(* CODESYS project SPT_NCI.library
   Version: 4.0.0
   Title: SPT NCI
   DefaultNamespace: SPT_NCI
   Placeholder: SPT NCI
   Company: Beckhoff Automation LLC

Project tree, tasks and I/O mapping:
  libraries: SPT Base Types, * (Beckhoff Automation LLC); SPT Event Logger, * (Beckhoff Automation LLC); Tc2_NCI, * (Beckhoff Automation GmbH); Tc2_Standard, * (Beckhoff Automation GmbH); Tc2_System, * (Beckhoff Automation GmbH); Tc3_EventLogger, * (Beckhoff Automation GmbH); Tc3_Module, * (Beckhoff Automation GmbH)
  DUTs/
    data type ST_NciBase_Command
    data type ST_NciBase_Config
    data type ST_NciBase_HMI
    data type ST_NciBase_Status
    data type ST_NciChannel
  FunctionBlocks/
    function block FB_Component_NciBase [ST]: Reset, CyclicLogic, BlockSearch, BuildNciGroup, ConfirmHsk, DissolveNciGroup, EnableRetrace, InterpreterStart, InterpreterStop, InterpreterStopOnPath, IsFastMFunction, LoadNciProgram, ResumeAfterEstop, RetraceBackward, RetraceForward, SetSearchOptionFlags, StepOnAfterBlocksearch, BlockSearchStartPosition, Channel, Deceleration, GetHskMFunction, GroupIsBuilt, InterpreterState, IsHandshake, Jerk, Override, ProgramPath, CreateEvents, HMICommunication, Monitoring, Q1AxisId, Q2AxisId, Q3AxisId, Q4AxisId, Q5AxisId, XAxisId, YAxisId, ZAxisId, Initialize
    function block FB_Component_NciParameterBase [ST]: Reset, CyclicLogic, CreateEvents, Channel, Initialize
    function block FB_Component_NciReadWriteRParameter [ST]: Reset, CyclicLogic, Monitoring, Read, Write
  Interfaces/
    interface I_NciBase: BlockSearch, BuildNciGroup, ConfirmHsk, DissolveNciGroup, EnableRetrace, InterpreterStart, InterpreterStop, InterpreterStopOnPath, IsFastMFunction, LoadNciProgram, ResumeAfterEstop, RetraceBackward, RetraceForward, SetSearchOptionFlags, StepOnAfterBlocksearch, BlockSearchStartPosition, Deceleration, GetHskMFunction, GroupIsBuilt, InterpreterState, IsHandshake, Jerk, Override, ProgramPath
    interface I_NciChannel: Channel
  Project Information/
    function F_GetCompany [ST]
    function F_GetTitle [ST]
    function F_GetVersion [ST]
  Utilities/
    function F_ADSErrorCodeExt [ST]
  Version/
    global variables Global_Version
  00000000-0000-0000-0000-000000000000|LICENSE
  LICENSE
*)

// DUTs/ST_NciBase_Command
TYPE ST_NciBase_Command :
	STRUCT
		BuildGroup		   : BOOL;
		DissolveGroup	   : BOOL;
		LoadNciProgram	   : BOOL;
		ItpStart		   : BOOL;
		ItpStop			   : BOOL;
		ItpEstopStopOnPath : BOOL;
		Resume			   : BOOL;
		SetOverride		   : BOOL;
		Override		   : UDINT; //Override in 0..1000000 (0..100%)
	END_STRUCT
END_TYPE

// DUTs/ST_NciBase_Config
TYPE ST_NciBase_Config :
	STRUCT
	END_STRUCT
END_TYPE

// DUTs/ST_NciBase_HMI
TYPE ST_NciBase_HMI :
	STRUCT
		Config	: ST_NciBase_Config;
		Command : ST_NciBase_Command;
		Status	: ST_NciBase_Status;
	END_STRUCT
END_TYPE

// DUTs/ST_NciBase_Status
TYPE ST_NciBase_Status :
	STRUCT
		NcToPlc : NCTOPLC_NCICHANNEL_REF;
	END_STRUCT
END_TYPE

// DUTs/ST_NciChannel
TYPE ST_NciChannel :
	STRUCT
		NcToPLC AT %I* : NCTOPLC_NCICHANNEL_REF;
		PlcToNc AT %Q* : PLCTONC_NCICHANNEL_REF;
	END_STRUCT
END_TYPE

// Version/Global_Version
{attribute 'TcGenerated'}
{attribute 'no-analysis'}
{attribute 'linkalways'}

// This function has been automatically generated from the project information.
VAR_GLOBAL CONSTANT
	{attribute 'const_non_replaced'}
	stLibVersion_SPT_NCI : ST_LibVersion := (iMajor := 4, iMinor := 0, iBuild := 0, iRevision := 0, nFlags := 0, sVersion := '4.0.0');
END_VAR

// FunctionBlocks/FB_Component_NciBase
FUNCTION_BLOCK FB_Component_NciBase EXTENDS FB_ComponentBase IMPLEMENTS I_NciBase
VAR
	// Channel connection
	NciChannel : ST_NciChannel;

	// Properties
	_ProgramPath		   : STRING := 'C:\TwinCAT\Mc\Nci\9999.nc';
	_XAxisId			   : UDINT	:= 0;
	_YAxisId			   : UDINT	:= 0;
	_ZAxisId			   : UDINT	:= 0;
	_Q1AxisId			   : UDINT	:= 0;
	_Q2AxisId			   : UDINT	:= 0;
	_Q3AxisId			   : UDINT	:= 0;
	_Q4AxisId			   : UDINT	:= 0;
	_Q5AxisId			   : UDINT	:= 0;
	_GroupIsBuilt		   : BOOL;
	_Jerk				   : LREAL;
	_Deceleration		   : LREAL;
	_BlockSearchOptionFlag : ST_ItpBlockSearchOptions := (bScanStartPos := TRUE);
	_StartPosition		   : ST_ItpBlockSearchStartPosition;

	// Internal Variables
	BuildGroup		 : CfgBuildExt3DGroup;
	DissolveGroup	 : CfgReconfigGroup;
	ResetNci		 : ItpResetEx2;
	LoadProgram		 : ItpLoadProgEx;
	StartStop		 : ItpStartStopEx;
	EStopOnPath		 : ItpEstopEx;
	StepOnAfterEStop : ItpStepOnAfterEStopEx;
	ResetFastMCode	 : ItpResetFastMFuncEx;
	ConfirmHandshake : ItpConfirmHsk;

	// Retrace functions
	EnableFeederBackup	: ItpEnableFeederBackup;
	RetraceMoveBackward : ItpRetraceMoveBackward;
	RetraceMoveForward	: ItpRetraceMoveForward;

	// Blocksearch
	InterpreterBlockSearch : ItpBlocksearch;
	BlockOn				   : ItpStepOnAfterBlocksearch;

	// HMI
	NciBase_HMI : ST_NciBase_HMI;

	// Alarms
	ComponentNciBaseAlarms : ARRAY[1..COMPONENT_NCI_BASE_ALARM_COUNT] OF FB_TcAlarm;
END_VAR

VAR CONSTANT
	COMPONENT_NCI_BASE_ALARM_COUNT : UDINT := 12;
END_VAR

// Clears error flags and error IDs for this component
METHOD PUBLIC Reset : BOOL
F_ClearAllEventsInClass(ComponentNciBaseAlarms);
_Error			  := FALSE;
_ErrorId		  := 0;
ResetNci.bExecute := TRUE;
Reset			  := SUPER^.Reset();
END_METHOD

// This method serves as the entry point for all underlying FB logic
METHOD PUBLIC CyclicLogic

// This method should be called cyclically by descendant function blocks by invoking SUPER^.CyclicLogic().  Alternatively, the contents of this method could be reimplemented entirely in which case a call to this method would not be necessary.
IF NOT _InitComplete THEN
	_InitComplete := Initialize();
	RETURN;
END_IF

(* NCI FBs *)

// Build NCI Group
BuildGroup(nGroupId := NciChannel.NcToPLC.GrpId, tTimeout := T#1S);
IF BuildGroup.bErr AND BuildGroup.bExecute THEN
	_GroupIsBuilt := FALSE;
	_Error		  := TRUE;
	_ErrorId	  := BuildGroup.nErrId;
END_IF

IF NOT BuildGroup.bBusy THEN
	BuildGroup.bExecute := FALSE;
END_IF

// Dissolve NCI Group
DissolveGroup(nGroupId := NciChannel.NcToPLC.GrpId, tTimeOut := T#1S);
IF DissolveGroup.bErr AND DissolveGroup.bExecute THEN
	_Error	 := TRUE;
	_ErrorId := DissolveGroup.nErrId;
END_IF

IF NOT DissolveGroup.bBusy THEN
	DissolveGroup.bExecute := FALSE;
END_IF

// Reset
ResetNci(sNciToPlc := NciChannel.NcToPlc, tTimeOut := T#1S);
IF ResetNci.bErr AND ResetNci.bExecute THEN
	_Error	 := TRUE;
	_ErrorId := ResetNci.nErrId;
END_IF

IF NOT ResetNci.bBusy THEN
	ResetNci.bExecute := FALSE;
END_IF

// Load Program
LoadProgram(sNciToPlc := NciChannel.NcToPLC,
			sPrg	  := _ProgramPath,
			nLength	  := INT_TO_UDINT(LEN(_ProgramPath)),
			tTimeOut  := T#1S);

IF LoadProgram.bErr AND LoadProgram.bExecute THEN
	_Error	 := TRUE;
	_ErrorId := LoadProgram.nErrId;
END_IF

IF NOT LoadProgram.bBusy THEN
	LoadProgram.bExecute := FALSE;
END_IF

// Start/Stop Interpreter
StartStop(sNciToPlc := NciChannel.NcToPLC, tTimeOut := T#1S);
IF StartStop.bErr AND (StartStop.bStop OR StartStop.bStart) THEN
	_Error	 := TRUE;
	_ErrorId := StartStop.nErrId;
END_IF

IF NOT StartStop.bBusy THEN
	StartStop.bStop	 := FALSE;
	StartStop.bStart := FALSE;
END_IF

//
EStopOnPath(sNciToPlc := NciChannel.NcToPLC,
			fDec	  := _Deceleration,
			fJerk	  := _Jerk,
			tTimeOut  := T#1S);

IF EStopOnPath.bErr AND EStopOnPath.bExecute THEN
	_Error	 := TRUE;
	_ErrorId := EStopOnPath.nErrId;
END_IF

IF NOT EStopOnPath.bBusy THEN
	EStopOnPath.bExecute := FALSE;
END_IF

StepOnAfterEStop(sNciToPlc := NciChannel.NcToPLC, tTimeOut := T#1S);
IF StepOnAfterEStop.bErr AND StepOnAfterEStop.bExecute THEN
	_Error	 := TRUE;
	_ErrorId := StepOnAfterEStop.nErrId;
END_IF

IF NOT StepOnAfterEStop.bBusy THEN
	StepOnAfterEStop.bExecute := FALSE;
END_IF

// Retracing
EnableFeederBackup(bEnable := TRUE, tTimeOut := T#1S, sNciToPlc := NciChannel.NcToPLC);
IF EnableFeederBackup.bErr AND EnableFeederBackup.bExecute THEN
	_Error	 := TRUE;
	_ErrorId := EnableFeederBackup.nErrId;
END_IF

IF NOT EnableFeederBackup.bBusy THEN
	EnableFeederBackup.bExecute := FALSE;
END_IF

RetraceMoveBackward(sNciToPlc := NciChannel.NcToPLC);
IF RetraceMoveBackward.bErr AND RetraceMoveBackward.bExecute THEN
	_Error	 := TRUE;
	_ErrorId := RetraceMoveBackward.nErrId;
END_IF

IF NOT RetraceMoveBackward.bBusy THEN
	RetraceMoveBackward.bExecute := FALSE;
END_IF

RetraceMoveForward(sNciToPlc := NciChannel.NcToPLC);
IF RetraceMoveForward.bErr AND RetraceMoveForward.bExecute THEN
	_Error	 := TRUE;
	_ErrorId := RetraceMoveForward.nErrId;
END_IF

IF NOT RetraceMoveForward.bBusy THEN
	RetraceMoveForward.bExecute := FALSE;
END_IF

// Blocksearch
InterpreterBlockSearch(sPrgName		  := _ProgramPath,
					   nPrgLength	  := INT_TO_UDINT(LEN(_ProgramPath)),
					   tTimeOut		  := T#5S,
					   sAxesList	  :=,
					   sOptions		  := _BlockSearchOptionFlag,
					   sStartPosition => _StartPosition,
					   sNciToPlc	  := NciChannel.NcToPLC);

IF InterpreterBlockSearch.bErr AND InterpreterBlockSearch.bExecute THEN
	_Error	 := TRUE;
	_ErrorId := InterpreterBlockSearch.nErrId;
END_IF

IF NOT InterpreterBlockSearch.bBusy THEN
	InterpreterBlockSearch.bExecute := FALSE;
END_IF

BlockOn(sNciToPlc := NciChannel.NcToPLC, tTimeOut := T#1S);
IF BlockOn.bErr AND BlockOn.bExecute THEN
	_Error	 := TRUE;
	_ErrorId := BlockOn.nErrId;
END_IF

IF NOT BlockOn.bBusy THEN
	BlockOn.bExecute := FALSE;
END_IF

// MCode
ResetFastMCode(sNciToPlc := NciChannel.NcToPLC, tTimeOut := T#1S);
ResetFastMCode.bExecute := FALSE;
ConfirmHandshake(sNciToPlc := NciChannel.NcToPlc, sPlcToNci := NciChannel.PlcToNc);
ConfirmHandshake.bExecute := FALSE;

// Busy
_Busy := ResetNci.bBusy OR DissolveGroup.bBusy OR BuildGroup.bBusy OR EnableFeederBackup.bBusy OR EStopOnPath.bBusy OR RetraceMoveForward.bBusy OR RetraceMoveBackward.bBusy OR InterpreterBlockSearch.bBusy OR BlockOn.bBusy;

// Call Super
SUPER^.CyclicLogic();
_CurrentAlarmSeverity := F_GetMaxSeverityRaised(Alarms := ComponentNciBaseAlarms, CurrentSeverity := _CurrentAlarmSeverity);
END_METHOD

METHOD BlockSearch : BOOL
VAR_INPUT
	BlockId			: UINT;
	BlockSearchMode : E_ItpBlockSearchMode;
	DryRunMode		: E_ItpDryRunMode;
	LineLength		: UDINT;
END_VAR
IF _Busy OR _Error THEN
	RETURN;
END_IF

InterpreterBlockSearch.nBlockId			:= BlockId;
InterpreterBlockSearch.eBlockSearchMode := BlockSearchMode;
InterpreterBlockSearch.eDryRunMode		:= DryRunMode;
InterpreterBlockSearch.fLength			:= LineLength;
InterpreterBlockSearch.bExecute			:= TRUE;
BlockSearch								:= TRUE;
END_METHOD

METHOD PUBLIC BuildNciGroup : BOOL
IF _Busy OR _Error THEN
	RETURN;
END_IF

BuildGroup.nXAxisId	 := _XAxisId;
BuildGroup.nYAxisId	 := _YAxisId;
BuildGroup.nZAxisId	 := _ZAxisId;
BuildGroup.nQ1AxisId := _Q1AxisId;
BuildGroup.nQ2AxisId := _Q2AxisId;
BuildGroup.nQ3AxisId := _Q3AxisId;
BuildGroup.nQ4AxisId := _Q4AxisId;
BuildGroup.nQ5AxisId := _Q5AxisId;
BuildGroup.bExecute	 := TRUE;
_GroupIsBuilt		 := TRUE;
BuildNciGroup		 := TRUE;
END_METHOD

METHOD ConfirmHsk : BOOL
VAR_INPUT
END_VAR
ConfirmHandshake.bExecute := TRUE;
ConfirmHsk				  := TRUE;
END_METHOD

METHOD PUBLIC DissolveNciGroup : BOOL
IF _Busy THEN
	RETURN;
END_IF

_GroupIsBuilt		   := FALSE;
DissolveGroup.bExecute := TRUE;
DissolveNciGroup	   := TRUE;
END_METHOD

METHOD EnableRetrace : BOOL
VAR_INPUT
END_VAR
IF _Busy OR _Error THEN
	RETURN;
END_IF

EnableFeederBackup.bExecute := TRUE;
EnableRetrace				:= TRUE;
END_METHOD

METHOD InterpreterStart : BOOL
IF _Busy OR _Error THEN
	RETURN;
END_IF

StartStop.bStart := TRUE;
InterpreterStart := TRUE;
END_METHOD

METHOD InterpreterStop : BOOL
StartStop.bStop := TRUE;
InterpreterStop := TRUE;
END_METHOD

METHOD InterpreterStopOnPath : BOOL
VAR_INPUT
END_VAR
EStopOnPath.bExecute  := TRUE;
InterpreterStopOnPath := TRUE;
END_METHOD

METHOD IsFastMFunction : BOOL
VAR_INPUT
	M		  : INT;
	AutoReset : BOOL; // Reset MCode at next cycle
END_VAR
IsFastMFunction := ItpIsFastMFunc(NFastMfuncNo := M, NciChannel.NcToPlc);
IF IsFastMfunction AND AutoReset THEN
	ResetFastMCode.nMFuncNo := TO_UINT(M);
	ResetFastMCode.bExecute := TRUE;
END_IF
END_METHOD

METHOD LoadNciProgram : BOOL
IF _Busy THEN
	RETURN;
END_IF

IF _ProgramPath = '' THEN
	TRACE('NCI Program can not be loaded, Path is empty!');
END_IF

LoadProgram.bExecute := TRUE;
LoadNciProgram		 := TRUE;
END_METHOD

// Resume after stop on patch (ItpEstopEx)
METHOD ResumeAfterEstop : BOOL
VAR_INPUT
END_VAR
IF _Busy OR _Error THEN
	RETURN;
END_IF

StepOnAfterEStop.bExecute := TRUE;
ResumeAfterEstop		  := TRUE;
END_METHOD

METHOD RetraceBackward : BOOL
VAR_INPUT
END_VAR
IF _Busy OR _Error THEN
	RETURN;
END_IF

RetraceMoveBackward.bExecute := TRUE;
RetraceBackward				 := TRUE;
END_METHOD

METHOD RetraceForward : BOOL
VAR_INPUT
END_VAR
IF _Busy OR _Error THEN
	RETURN;
END_IF

RetraceMoveForward.bExecute := TRUE;
RetraceForward				:= TRUE;
END_METHOD

METHOD SetSearchOptionFlags
VAR_INPUT
	IsRetrace		  : BOOL;
	IsRetraceBackward : BOOL;
	ScanStartPos	  : BOOL;
END_VAR
_BlockSearchOptionFlag.bIsRetrace		:= IsRetrace;
_BlockSearchOptionFlag.bRetraceBackward := IsRetraceBackward;
_BlockSearchOptionFlag.bScanStartPos	:= ScanStartPos;
END_METHOD

METHOD StepOnAfterBlocksearch : BOOL
VAR_INPUT
END_VAR
IF _Busy OR _Error THEN
	RETURN;
END_IF

BlockOn.bExecute	   := TRUE;
StepOnAfterBlocksearch := TRUE;
END_METHOD

PROPERTY BlockSearchStartPosition : ST_ItpBlockSearchStartPosition
GET
BlockSearchStartPosition := _StartPosition;
END_GET
END_PROPERTY

PROPERTY Channel : REFERENCE TO ST_NciChannel
GET
Channel REF= NciChannel;
END_GET
END_PROPERTY

PROPERTY Deceleration : LREAL
SET
_Deceleration := Deceleration;
END_SET
END_PROPERTY

PROPERTY GetHskMFunction : INT
GET
GetHskMFunction := ItpGetHskMFunc(NciChannel.NcToPLC);
END_GET
END_PROPERTY

PROPERTY GroupIsBuilt : BOOL
GET
GroupIsBuilt := _GroupIsBuilt;
END_GET
END_PROPERTY

// Use to query e.g. Tc2_NCI.NCI_INTERPRETER_READY
PROPERTY InterpreterState : UINT
GET
InterpreterState := NciChannel.NcToPLC.ItpState;
END_GET
END_PROPERTY

PROPERTY IsHandshake : BOOL
GET
IsHandshake := ItpIsHskMFunc(NciChannel.NcToPLC);
END_GET
END_PROPERTY

PROPERTY Jerk : LREAL
SET
_Jerk := Jerk;
END_SET
END_PROPERTY

// Override in 0..1000000 //Assigns override to all channel overrides, individual access via property channel.
PROPERTY Override : UDINT
SET
IF Override < 0 THEN
	NciChannel.PlcToNc.ChnAxesOvr	 := 0;
	NciChannel.PlcToNc.ChnSpindleOvr := 0;
ELSIF Override > 1_000_000 THEN
	NciChannel.PlcToNc.ChnAxesOvr	 := 1_000_000;
	NciChannel.PlcToNc.ChnSpindleOvr := 1_000_000;
ELSE
	NciChannel.PlcToNc.ChnAxesOvr	 := Override;
	NciChannel.PlcToNc.ChnSpindleOvr := Override;
END_IF
END_SET
END_PROPERTY

PROPERTY ProgramPath : STRING
GET
ProgramPath := _ProgramPath;
END_GET
SET
_ProgramPath := ProgramPath;
END_SET
END_PROPERTY

// Initializes event function blocks using this components's name
METHOD PROTECTED CreateEvents

// This method is called by Initialize() as required
SUPER^.CreateEvents();
F_CreateAllEventsInClass(Alarms		:= ComponentNciBaseAlarms,
						 ClassSize	:= SIZEOF(TC_EVENTS.NciAlarms),
						 pInitEvent := ADR(TC_EVENTS.NciAlarms.InitReferenceEvent),
						 Prefix		:= _Name);
END_METHOD

// Provides interlocks for HMI control and updates HMI status information for this component
METHOD PROTECTED HMICommunication
// This method is called cyclically by CyclicLogic()
VAR_INST
	HMICommandNciBase_RT : R_TRIG;
END_VAR
SUPER^.HMICommunication();
HMICommandNciBase_RT(CLK := (ComponentBase_HMI.Status.HMIControlAvailable AND NOT HMICommandActive_Base) AND (NciBase_HMI.Command.BuildGroup XOR NciBase_HMI.Command.DissolveGroup XOR NciBase_HMI.Command.LoadNciProgram XOR NciBase_HMI.Command.ItpStart XOR NciBase_HMI.Command.ItpStop XOR NciBase_Hmi.Command.ItpEstopStopOnPath XOR NciBase_Hmi.Command.Resume));

//Desendant components should observe this to interlock HMI commands
HMICommandActive_Descendant := ComponentBase_HMI.Status.HMIControlAvailable AND (NciBase_HMI.Command.BuildGroup OR NciBase_HMI.Command.DissolveGroup OR NciBase_HMI.Command.LoadNciProgram OR NciBase_HMI.Command.ItpStart OR NciBase_HMI.Command.ItpStop OR NciBase_Hmi.Command.ItpEstopStopOnPath OR NciBase_Hmi.Command.Resume);
IF HMICommandNciBase_RT.Q THEN
	IF NciBase_HMI.Command.BuildGroup THEN
		BuildNciGroup();
	END_IF

	IF NciBase_HMI.Command.DissolveGroup THEN
		DissolveNciGroup();
	END_IF

	IF NciBase_HMI.Command.LoadNciProgram THEN
		LoadNciProgram();
	END_IF

	IF NciBase_HMI.Command.ItpStart THEN
		InterpreterStart();
	END_IF

	IF NciBase_HMI.Command.ItpStop THEN
		InterpreterStop();
	END_IF

	IF NciBase_Hmi.Command.ItpEstopStopOnPath THEN
		InterpreterStopOnPath();
	END_IF

	IF NciBase_Hmi.Command.Resume THEN
		ResumeAfterEstop();
	END_IF
END_IF

NciBase_HMI.Command.BuildGroup		   := FALSE;
NciBase_HMI.Command.DissolveGroup	   := FALSE;
NciBase_HMI.Command.LoadNciProgram	   := FALSE;
NciBase_HMI.Command.ItpStart		   := FALSE;
NciBase_HMI.Command.ItpStop			   := FALSE;
NciBase_Hmi.Command.ItpEstopStopOnPath := FALSE;
NciBase_Hmi.Command.Resume			   := FALSE;

// Set Override
IF NciBase_Hmi.Command.SetOverride THEN
	Override						:= NciBase_Hmi.Command.Override;
	NciBase_Hmi.Command.SetOverride := FALSE;
END_IF

// Status
NciBase_Hmi.Status.NcToPlc := NciChannel.NcToPlc;
END_METHOD

// Provides basic error detection and event handling for this component
METHOD PROTECTED Monitoring
VAR_INST
	RTrigError	: R_TRIG; // Error active - Error Bit remains On in NCI Fbs until new command is issued
	TempMessage : STRING;
END_VAR

// This method is called cyclically by CyclicLogic()
SUPER^.Monitoring();
RTrigError(CLK := _Error);
IF RTrigError.Q THEN
	// Build Group
	IF BuildGroup.bErr AND NOT ComponentNciBaseAlarms[E_NciAlarms.BuildGroup].bRaised THEN
		RaiseAlarmWithStrings(ComponentNciBaseAlarms[E_NciAlarms.BuildGroup], F_ADSErrorCodeExt(_ErrorId), '');
	END_IF

	// Load Program
	IF LoadProgram.bErr AND NOT ComponentNciBaseAlarms[E_NciAlarms.LoadProgram].bRaised THEN
		RaiseAlarmWithStrings(ComponentNciBaseAlarms[E_NciAlarms.LoadProgram], F_ADSErrorCodeExt(_ErrorId), '');
	END_IF

	// Start/ Stop
	IF EStopOnPath.bErr AND NOT ComponentNciBaseAlarms[E_NciAlarms.StopOnPath].bRaised THEN
		RaiseAlarmWithStrings(ComponentNciBaseAlarms[E_NciAlarms.StopOnPath], F_ADSErrorCodeExt(_ErrorId), '');
	END_IF

	IF StartStop.bErr AND NOT ComponentNciBaseAlarms[E_NciAlarms.StartStop].bRaised THEN
		RaiseAlarmWithStrings(ComponentNciBaseAlarms[E_NciAlarms.StartStop], F_ADSErrorCodeExt(_ErrorId), '');
	END_IF

	IF StepOnAfterEStop.bErr AND NOT ComponentNciBaseAlarms[E_NciAlarms.StepOnAfterEStop].bRaised THEN
		RaiseAlarmWithStrings(ComponentNciBaseAlarms[E_NciAlarms.StepOnAfterEStop], F_ADSErrorCodeExt(_ErrorId), '');
	END_IF

	// Retracing
	IF EnableFeederBackup.bErr AND NOT ComponentNciBaseAlarms[E_NciAlarms.EnableFeederBackup].bRaised THEN
		RaiseAlarmWithStrings(ComponentNciBaseAlarms[E_NciAlarms.EnableFeederBackup], F_ADSErrorCodeExt(_ErrorId), '');
	END_IF

	IF RetraceMoveBackward.bErr AND NOT ComponentNciBaseAlarms[E_NciAlarms.RetraceMoveBackward].bRaised THEN
		RaiseAlarmWithStrings(ComponentNciBaseAlarms[E_NciAlarms.RetraceMoveBackward], F_ADSErrorCodeExt(_ErrorId), '');
	END_IF

	IF RetraceMoveForward.bErr AND NOT ComponentNciBaseAlarms[E_NciAlarms.RetraceMoveForward].bRaised THEN
		RaiseAlarmWithStrings(ComponentNciBaseAlarms[E_NciAlarms.RetraceMoveForward], F_ADSErrorCodeExt(_ErrorId), '');
	END_IF

	// Blocksearch
	IF InterpreterBlockSearch.bErr AND NOT ComponentNciBaseAlarms[E_NciAlarms.InterpreterBlockSearch].bRaised THEN
		RaiseAlarmWithStrings(ComponentNciBaseAlarms[E_NciAlarms.InterpreterBlockSearch], F_ADSErrorCodeExt(_ErrorId), '');
	END_IF

	IF BlockOn.bErr AND NOT ComponentNciBaseAlarms[E_NciAlarms.BlockOn].bRaised THEN
		RaiseAlarmWithStrings(ComponentNciBaseAlarms[E_NciAlarms.BlockOn], F_ADSErrorCodeExt(_ErrorId), '');
	END_IF
END_IF

IF (THIS^.InterpreterState = Tc2_NCI.NCI_INTERPRETER_INITFAILED) OR (THIS^.InterpreterState = Tc2_NCI.NCI_INTERPRETER_ABORTED) OR (THIS^.InterpreterState = Tc2_NCI.NCI_INTERPRETER_FAULT) THEN
	IF THIS^.InterpreterState = Tc2_NCI.NCI_INTERPRETER_INITFAILED THEN
		TempMessage := 'INITFAILED';
	ELSIF THIS^.InterpreterState = Tc2_NCI.NCI_INTERPRETER_ABORTED THEN
		TempMessage := 'ABORTED';
	ELSIF THIS^.InterpreterState = Tc2_NCI.NCI_INTERPRETER_FAULT THEN
		TempMessage := 'FAULT';
	END_IF

	IF NOT ComponentNciBaseAlarms[E_NciAlarms.InterpreterError].bRaised THEN
		RaiseAlarmWithStrings(ComponentNciBaseAlarms[E_NciAlarms.InterpreterError], F_ADSErrorCodeExt(NciChannel.NcToPLC.ErrorCode), TempMessage);
	END_IF
END_IF
END_METHOD

PROPERTY Q1AxisId : UDINT
GET
Q1AxisId := _Q1AxisId;
END_GET
SET
_Q1AxisId := Q1AxisId;
END_SET
END_PROPERTY

PROPERTY Q2AxisId : UDINT
GET
Q2AxisId := _Q2AxisId;
END_GET
SET
_Q2AxisId := Q2AxisId;
END_SET
END_PROPERTY

PROPERTY Q3AxisId : UDINT
GET
Q3AxisId := _Q3AxisId;
END_GET
SET
_Q3AxisId := Q3AxisId;
END_SET
END_PROPERTY

PROPERTY Q4AxisId : UDINT
GET
Q4AxisId := _Q4AxisId;
END_GET
SET
_Q4AxisId := Q4AxisId;
END_SET
END_PROPERTY

PROPERTY Q5AxisId : UDINT
GET
Q5AxisId := _Q5AxisId;
END_GET
SET
_Q5AxisId := Q5AxisId;
END_SET
END_PROPERTY

PROPERTY XAxisId : UDINT
GET
XAxisId := _XAxisId;
END_GET
SET
_XAxisId := XAxisId;
END_SET
END_PROPERTY

PROPERTY YAxisId : UDINT
GET
YAxisId := _YAxisId;
END_GET
SET
_YAxisId := YAxisId;
END_SET
END_PROPERTY

PROPERTY ZAxisId : UDINT
GET
ZAxisId := _ZAxisId;
END_GET
SET
_ZAxisId := ZAxisId;
END_SET
END_PROPERTY

// Basic component initialization logic
METHOD PROTECTED Initialize : BOOL;

// This method is called by CyclicLogic() as required
IF F_GetMappingStatus(ADR(NciChannel.NcToPLC), SIZEOF(NciChannel.NcToPLC)) = EPlcMappingStatus.MS_Unmapped THEN
	TRACE('NcToPLC not mapped!');
	_Error	 := TRUE;
	_ErrorId := 1;
	RETURN;
END_IF

IF F_GetMappingStatus(ADR(NciChannel.PlcToNc), SIZEOF(NciChannel.PlcToNc)) = EPlcMappingStatus.MS_Unmapped THEN
	TRACE('PlcToNc not mapped!');
	_Error	 := TRUE;
	_ErrorId := 2;
	RETURN;
END_IF

Initialize := SUPER^.Initialize();
END_METHOD

END_FUNCTION_BLOCK

// Interfaces/I_NciBase
INTERFACE I_NciBase EXTENDS I_BaseFB, I_NciChannel

METHOD BlockSearch : BOOL
VAR_INPUT
	BlockId			: UINT;
	BlockSearchMode : E_ItpBlockSearchMode;
	DryRunMode		: E_ItpDryRunMode;
	LineLength		: UDINT;
END_VAR
END_METHOD

METHOD PUBLIC BuildNciGroup : BOOL
END_METHOD

METHOD ConfirmHsk : BOOL
VAR_INPUT
END_VAR
END_METHOD

METHOD PUBLIC DissolveNciGroup : BOOL
END_METHOD

METHOD EnableRetrace : BOOL
VAR_INPUT
END_VAR
END_METHOD

METHOD InterpreterStart : BOOL
END_METHOD

METHOD InterpreterStop : BOOL
END_METHOD

METHOD InterpreterStopOnPath : BOOL
VAR_INPUT
END_VAR
END_METHOD

METHOD IsFastMFunction : BOOL
VAR_INPUT
	M		  : INT;
	AutoReset : BOOL; // Reset MCode at next cycle
END_VAR
END_METHOD

METHOD LoadNciProgram : BOOL
END_METHOD

// Resume after stop on patch (ItpEstopEx)
METHOD ResumeAfterEstop : BOOL
VAR_INPUT
END_VAR
END_METHOD

METHOD RetraceBackward : BOOL
VAR_INPUT
END_VAR
END_METHOD

METHOD RetraceForward : BOOL
VAR_INPUT
END_VAR
END_METHOD

METHOD SetSearchOptionFlags
VAR_INPUT
	IsRetrace		  : BOOL;
	IsRetraceBackward : BOOL;
	ScanStartPos	  : BOOL;
END_VAR
END_METHOD

METHOD StepOnAfterBlocksearch : BOOL
VAR_INPUT
END_VAR
END_METHOD

PROPERTY BlockSearchStartPosition : ST_ItpBlockSearchStartPosition
GET
END_GET
END_PROPERTY

PROPERTY Deceleration : LREAL
SET
END_SET
END_PROPERTY

PROPERTY GetHskMFunction : INT
GET
END_GET
END_PROPERTY

PROPERTY GroupIsBuilt : BOOL
GET
END_GET
END_PROPERTY

// Use to query e.g. Tc2_NCI.NCI_INTERPRETER_READY
PROPERTY InterpreterState : UINT
GET
END_GET
END_PROPERTY

PROPERTY IsHandshake : BOOL
GET
END_GET
END_PROPERTY

PROPERTY Jerk : LREAL
SET
END_SET
END_PROPERTY

// Override in 0..1000000 //Assigns override to all channel overrides, individual access via property channel.
PROPERTY Override : UDINT
SET
END_SET
END_PROPERTY

PROPERTY ProgramPath : STRING
GET
END_GET
SET
END_SET
END_PROPERTY

END_INTERFACE

// Interfaces/I_NciChannel
INTERFACE I_NciChannel

PROPERTY Channel : REFERENCE TO ST_NciChannel
GET
END_GET
END_PROPERTY

END_INTERFACE

// Utilities/F_ADSErrorCodeExt
// Extended version of ADS Error Code with "Further Error codes" incl. Kinematic Error Codes
FUNCTION F_ADSErrorCodeExt : STRING(255)
VAR_INPUT
	ErrorId : UDINT;
END_VAR

VAR
END_VAR

CASE ErrorId OF
	// Global Error Codes 

	// 0 - 30					
	0:
		F_ADSErrorCodeExt := 'No error id found';

	1:
		F_ADSErrorCodeExt := 'Internal error.';

	2:
		F_ADSErrorCodeExt := 'No real time.';

	3:
		F_ADSErrorCodeExt := 'Allocation locked – memory error.';

	4:
		F_ADSErrorCodeExt := 'Mailbox full – the ADS message could not be sent. Reducing the number of ADS messages per cycle will help.';

	5:
		F_ADSErrorCodeExt := 'Wrong HMSG.';

	6:
		F_ADSErrorCodeExt := 'Target port not found – ADS server is not started or is not reachable.';

	7:
		F_ADSErrorCodeExt := 'Target computer not found – AMS route was not found.';

	8:
		F_ADSErrorCodeExt := 'Unknown command ID.';

	9:
		F_ADSErrorCodeExt := 'Invalid task ID.';

	10:
		F_ADSErrorCodeExt := 'No IO.';

	11:
		F_ADSErrorCodeExt := 'Unknown AMS command.';

	12:
		F_ADSErrorCodeExt := 'Win32 error.';

	13:
		F_ADSErrorCodeExt := 'Port not connected.';

	14:
		F_ADSErrorCodeExt := 'Invalid AMS length.';

	15:
		F_ADSErrorCodeExt := 'Invalid AMS Net ID.';

	16:
		F_ADSErrorCodeExt := 'Installation level is too low –TwinCAT 2 license error.';

	17:
		F_ADSErrorCodeExt := 'No debugging available.';

	18:
		F_ADSErrorCodeExt := 'Port disabled – TwinCAT system service not started.';

	19:
		F_ADSErrorCodeExt := 'Port already connected.';

	20:
		F_ADSErrorCodeExt := 'AMS Sync Win32 error.';

	21:
		F_ADSErrorCodeExt := 'AMS Sync Timeout.';

	22:
		F_ADSErrorCodeExt := 'AMS Sync error.';

	23:
		F_ADSErrorCodeExt := 'No index map for AMS Sync available.';

	24:
		F_ADSErrorCodeExt := 'Invalid AMS port.';

	25:
		F_ADSErrorCodeExt := 'No memory.';

	26:
		F_ADSErrorCodeExt := 'TCP send error.';

	27:
		F_ADSErrorCodeExt := 'Host unreachable.';

	28:
		F_ADSErrorCodeExt := 'Invalid AMS fragment.';

	29:
		F_ADSErrorCodeExt := 'TLS send error – secure ADS connection failed.';

	30:
		F_ADSErrorCodeExt := 'Access denied – secure ADS access denied.';

		// Router Error Codes 

	// 1280 - 1293					
	1280:
		F_ADSErrorCodeExt := 'Locked memory cannot be allocated.';

	1281:
		F_ADSErrorCodeExt := 'The router memory size could not be changed.';

	1282:
		F_ADSErrorCodeExt := 'The mailbox has reached the maximum number of possible messages.';

	1283:
		F_ADSErrorCodeExt := 'The Debug mailbox has reached the maximum number of possible messages.';

	1284:
		F_ADSErrorCodeExt := 'The port type is unknown.';

	1285:
		F_ADSErrorCodeExt := 'The router is not initialized.';

	1286:
		F_ADSErrorCodeExt := 'The port number is already assigned.';

	1287:
		F_ADSErrorCodeExt := 'The port is not registered.';

	1288:
		F_ADSErrorCodeExt := 'The maximum number of ports has been reached.';

	1289:
		F_ADSErrorCodeExt := 'The port is invalid.';

	1290:
		F_ADSErrorCodeExt := 'The router is not active.';

	1291:
		F_ADSErrorCodeExt := 'The mailbox has reached the maximum number for fragmented messages.';

	1292:
		F_ADSErrorCodeExt := 'A fragment timeout has occurred.';

	1293:
		F_ADSErrorCodeExt := 'The port is removed.';

		// General Error Codes 

	// 1792 - 1877							
	1792:
		F_ADSErrorCodeExt := 'General device error.';

	1793:
		F_ADSErrorCodeExt := 'Service is not supported by the server.';

	1794:
		F_ADSErrorCodeExt := 'Invalid index group.';

	1795:
		F_ADSErrorCodeExt := 'Invalid index offset.';

	1796:
		F_ADSErrorCodeExt := 'Reading or writing not permitted.';

	1797:
		F_ADSErrorCodeExt := 'Parameter size not correct.';

	1798:
		F_ADSErrorCodeExt := 'Invalid data values.';

	1799:
		F_ADSErrorCodeExt := 'Device is not ready to operate.';

	1800:
		F_ADSErrorCodeExt := 'Device is busy.';

	1801:
		F_ADSErrorCodeExt := 'Invalid operating system context. This can result from use of ADS blocks in different tasks. It may be possible to resolve this through multitasking synchronization in the PLC.';

	1802:
		F_ADSErrorCodeExt := 'Insufficient memory.';

	1803:
		F_ADSErrorCodeExt := 'Invalid parameter values.';

	1804:
		F_ADSErrorCodeExt := 'Not found (files, ...).';

	1805:
		F_ADSErrorCodeExt := 'Syntax error in file or command.';

	1806:
		F_ADSErrorCodeExt := 'Objects do not match.';

	1807:
		F_ADSErrorCodeExt := 'Object already exists.';

	1808:
		F_ADSErrorCodeExt := 'Symbol not found.';

	1809:
		F_ADSErrorCodeExt := 'Invalid symbol version. This can occur due to an online change. Create a new handle.';

	1810:
		F_ADSErrorCodeExt := 'Device (server) is in invalid state.';

	1811:
		F_ADSErrorCodeExt := 'AdsTransMode not supported.';

	1812:
		F_ADSErrorCodeExt := 'Notification handle is invalid.';

	1813:
		F_ADSErrorCodeExt := 'Notification client not registered.';

	1814:
		F_ADSErrorCodeExt := 'No further handle available.';

	1815:
		F_ADSErrorCodeExt := 'Notification size too large.';

	1816:
		F_ADSErrorCodeExt := 'Device not initialized.';

	1817:
		F_ADSErrorCodeExt := 'Device has a timeout.';

	1818:
		F_ADSErrorCodeExt := 'Interface query failed.';

	1819:
		F_ADSErrorCodeExt := 'Wrong interface requested.';

	1820:
		F_ADSErrorCodeExt := 'Class ID is invalid.';

	1821:
		F_ADSErrorCodeExt := 'Object ID is invalid.';

	1822:
		F_ADSErrorCodeExt := 'Request pending.';

	1823:
		F_ADSErrorCodeExt := 'Request is aborted.';

	1824:
		F_ADSErrorCodeExt := 'Signal warning.';

	1825:
		F_ADSErrorCodeExt := 'Invalid array index.';

	1826:
		F_ADSErrorCodeExt := 'Symbol not active.';

	1827:
		F_ADSErrorCodeExt := 'Access denied.';

	1828:
		F_ADSErrorCodeExt := 'Missing license.';

	1829:
		F_ADSErrorCodeExt := 'License expired.';

	1830:
		F_ADSErrorCodeExt := 'License exceeded.';

	1831:
		F_ADSErrorCodeExt := 'Invalid license.';

	1832:
		F_ADSErrorCodeExt := 'License problem: System ID is invalid.';

	1833:
		F_ADSErrorCodeExt := 'License not limited in time.';

	1834:
		F_ADSErrorCodeExt := 'Licensing problem: time in the future.';

	1835:
		F_ADSErrorCodeExt := 'License period too long.';

	1836:
		F_ADSErrorCodeExt := 'Exception at system startup.';

	1837:
		F_ADSErrorCodeExt := 'License file read twice.';

	1838:
		F_ADSErrorCodeExt := 'Invalid signature.';

	1839:
		F_ADSErrorCodeExt := 'Invalid certificate.';

	1840:
		F_ADSErrorCodeExt := 'Public key not known from OEM.';

	1841:
		F_ADSErrorCodeExt := 'License not valid for this system ID.';

	1842:
		F_ADSErrorCodeExt := 'Demo license prohibited.';

	1843:
		F_ADSErrorCodeExt := 'Invalid function ID.';

	1844:
		F_ADSErrorCodeExt := 'Outside the valid range.';

	1845:
		F_ADSErrorCodeExt := 'Invalid alignment.';

	1846:
		F_ADSErrorCodeExt := 'Invalid platform level.';

	1847:
		F_ADSErrorCodeExt := 'Context – forward to passive level.';

	1848:
		F_ADSErrorCodeExt := 'Context – forward to dispatch level.';

	1849:
		F_ADSErrorCodeExt := 'Context – forward to real time.';

	1856:
		F_ADSErrorCodeExt := 'Client error.';

	1857:
		F_ADSErrorCodeExt := 'Service contains an invalid parameter.';

	1858:
		F_ADSErrorCodeExt := 'Polling list is empty.';

	1859:
		F_ADSErrorCodeExt := 'Var connection already in use.';

	1860:
		F_ADSErrorCodeExt := 'The called ID is already in use.';

	1861:
		F_ADSErrorCodeExt := 'Timeout has occurred – the remote terminal is not responding in the specified ADS timeout. The route setting of the remote terminal may be configured incorrectly.';

	1862:
		F_ADSErrorCodeExt := 'Error in Win32 subsystem.';

	1863:
		F_ADSErrorCodeExt := 'Invalid client timeout value.';

	1864:
		F_ADSErrorCodeExt := 'Port not open.';

	1865:
		F_ADSErrorCodeExt := 'No AMS address.';

	1872:
		F_ADSErrorCodeExt := 'Internal error in Ads sync.';

	1873:
		F_ADSErrorCodeExt := 'Hash table overflow.';

	1874:
		F_ADSErrorCodeExt := 'Key not found in the table.';

	1875:
		F_ADSErrorCodeExt := 'No symbols in the cache.';

	1876:
		F_ADSErrorCodeExt := 'Invalid response received.';

	1877:
		F_ADSErrorCodeExt := 'Sync Port is locked.';

		// RTime Error Codes 

	// 4096 - 4122								
	4096:
		F_ADSErrorCodeExt := 'Internal error in the real-time system.';

	4097:
		F_ADSErrorCodeExt := 'Timer value is not valid.';

	4098:
		F_ADSErrorCodeExt := 'Task pointer has the invalid value 0 (zero).';

	4099:
		F_ADSErrorCodeExt := 'Stack pointer has the invalid value 0 (zero).';

	4100:
		F_ADSErrorCodeExt := 'The request task priority is already assigned.';

	4101:
		F_ADSErrorCodeExt := 'No free TCB (Task Control Block) available. The maximum number of TCBs is 64.';

	4102:
		F_ADSErrorCodeExt := 'No free semaphores available. The maximum number of semaphores is 64.';

	4103:
		F_ADSErrorCodeExt := 'No free space available in the queue. The maximum number of positions in the queue is 64.';

	4109:
		F_ADSErrorCodeExt := 'An external synchronization interrupt is already applied.';

	4110:
		F_ADSErrorCodeExt := 'No external sync interrupt applied.';

	4111:
		F_ADSErrorCodeExt := 'Application of the external synchronization interrupt has failed.';

	4112:
		F_ADSErrorCodeExt := 'Call of a service function in the wrong context';

	4119:
		F_ADSErrorCodeExt := 'Intel VT-x extension is not supported.';

	4120:
		F_ADSErrorCodeExt := 'Intel VT-x extension is not enabled in the BIOS.';

	4121:
		F_ADSErrorCodeExt := 'Missing function in Intel VT-x extension.';

	4122:
		F_ADSErrorCodeExt := 'Activation of Intel VT-x fails.';

		// TCP Winsock Error Codes 

	// 10060 - 10065									
	10060:
		F_ADSErrorCodeExt := 'A connection timeout has occurred. Error WHILE establishing the connection.';

	10061:
		F_ADSErrorCodeExt := 'Connection refused. No connection could be established because the target computer has explicitly rejected it.';

	10065:
		F_ADSErrorCodeExt := 'No route to host - a socket operation referred to an unavailable host.';

		// NC - General Error Codes 

	// 16384 - 16497
	16384:
		F_ADSErrorCodeExt := 'Internal system error in the NC on ring 0, no further details.';

	16385:
		F_ADSErrorCodeExt := 'The ring-0 memory management is not providing the required memory.';

	16386:
		F_ADSErrorCodeExt := 'Error while loading the Nc retain data.';

	16387:
		F_ADSErrorCodeExt := 'Parameter for Monitoring the NC Setpoint Issuing is Invalid.';

	16388:
		F_ADSErrorCodeExt := 'External Error.';

	16400:
		F_ADSErrorCodeExt := 'Channel identifier not allowed.';

	16401:
		F_ADSErrorCodeExt := 'Group identifier not allowed.';

	16402:
		F_ADSErrorCodeExt := 'Axis identifier not allowed.';

	16403:
		F_ADSErrorCodeExt := 'Encoder identifier not allowed.';

	16404:
		F_ADSErrorCodeExt := 'Controller identifier not allowed.';

	16405:
		F_ADSErrorCodeExt := 'Drive identifier not allowed.';

	16406:
		F_ADSErrorCodeExt := 'Table identifier not allowed.';

	16416:
		F_ADSErrorCodeExt := 'No PLC-axis interface during creation of an axis.';

	16417:
		F_ADSErrorCodeExt := 'No axis-PLC interface during creation of an axis.';

	16418:
		F_ADSErrorCodeExt := 'No encoder-I/O interface during creation of an axis.';

	16419:
		F_ADSErrorCodeExt := 'No I/O-encoder interface during creation of an axis.';

	16420:
		F_ADSErrorCodeExt := 'No drive-I/O interface during creation of an axis.';

	16421:
		F_ADSErrorCodeExt := 'No I/O-drive interface during creation of an axis.';

	16432:
		F_ADSErrorCodeExt := 'Coupling type not allowed. Unacceptable master/slave coupling type.';

	16433:
		F_ADSErrorCodeExt := 'Axis type not allowed. Unacceptable type specification during creation of an axis.';

	16434:
		F_ADSErrorCodeExt := 'Unknown Channel Type.';

	16448:
		F_ADSErrorCodeExt := 'Axis is not suitable for the intended purpose.';

	16464:
		F_ADSErrorCodeExt := 'Channel not ready for operation.';

	16465:
		F_ADSErrorCodeExt := 'Group not ready for operation.';

	16466:
		F_ADSErrorCodeExt := 'Axis not ready for operation.';

	16480:
		F_ADSErrorCodeExt := 'The channel that is to be created already exists.';

	16481:
		F_ADSErrorCodeExt := 'The group that is to be created already exists.';

	16482:
		F_ADSErrorCodeExt := 'The axis that is to be created already exists.';

	16483:
		F_ADSErrorCodeExt := 'The table that is to be created already exists, resp. it is tried internally to use an already existing table id ( e.g. for the universal flying saw).';

	16496:
		F_ADSErrorCodeExt := 'The location within the channel specified for an axis is not allowed.';

	16497:
		F_ADSErrorCodeExt := 'The location within the group specified for an axis is not allowed.';

		// NC - Channel Error Codes 

	// 16641 - 16756)					
	16641:
		F_ADSErrorCodeExt := 'Group index not allowed.';

	16642:
		F_ADSErrorCodeExt := 'The pointer to the group is invalid.';

	16643:
		F_ADSErrorCodeExt := 'No process image. It is not possible to exchange data with the PLC.';

	16644:
		F_ADSErrorCodeExt := 'Unacceptable M-function (not 0...159) detected at the execution level.';

	16645:
		F_ADSErrorCodeExt := 'No more system memory is available. This is usually the result of another error.';

	16646:
		F_ADSErrorCodeExt := 'The function is not presently available, because a similar function is already being processed.';

	16647:
		F_ADSErrorCodeExt := 'A requested function or command is not supported by the channel.';

	16648:
		F_ADSErrorCodeExt := 'Parameters to start the channel (TwinCAT-Start) are invalid.';

	16649:
		F_ADSErrorCodeExt := 'Channel function/command not executable. e.g. interpreter start is not executable because the channel is already busy, no program is loaded or in an error state.';

	16650:
		F_ADSErrorCodeExt := 'ItpGoAhead not executable. because the interpreter is not executing a decoder stop.';

	16656:
		F_ADSErrorCodeExt := 'The specified file does not exist.';

	16657:
		F_ADSErrorCodeExt := 'Syntax error during loading.';

	16658:
		F_ADSErrorCodeExt := 'Syntax error during interpretation.';

	16659:
		F_ADSErrorCodeExt := 'The NC has found a missing subroutine while loading.';

	16660:
		F_ADSErrorCodeExt := 'The capacity of the interpreter loading buffer has been exceeded.';

	16661:
		F_ADSErrorCodeExt := 'Symbolic - reserved';

	16662:
		F_ADSErrorCodeExt := 'Symbolic - reserved';

	16663:
		F_ADSErrorCodeExt := 'Subroutine incomplete. Header of subroutine is missing';

	16664:
		F_ADSErrorCodeExt := 'Error while loading the NC program. The maximum number of loadable NC programs has been reached. Possible cause: Too many sub-programs were loaded from a main program.';

	16665:
		F_ADSErrorCodeExt := 'Error while loading the NC program. The program name is too long.';

	16672:
		F_ADSErrorCodeExt := 'Divide by zero.';

	16673:
		F_ADSErrorCodeExt := 'Invalid circle parameterization. The specified circle cannot be calculated.';

	16674:
		F_ADSErrorCodeExt := 'Invalid FPU-Operation. e.g. by calculating the square root of a negative number.';

	16688:
		F_ADSErrorCodeExt := 'Stack overflow: subroutines. The NC encountered a stack overflow during execution: too many subroutine levels.';

	16689:
		F_ADSErrorCodeExt := 'Stack underflow: subroutines. The NC encountered a stack underflow during execution: too many subroutine return commands. Note: A main program must not end with a return command.';

	16690:
		F_ADSErrorCodeExt := 'Stack overflow: arithmetic unit. The NC encountered a stack overflow during execution: The calculation is too complex, or has not been correctly written.';

	16691:
		F_ADSErrorCodeExt := 'Stack underflow: arithmetic unit. The NC encountered a stack underflow during execution: The calculation is too complex, or has not been correctly written.';

	16704:
		F_ADSErrorCodeExt := 'Register index not allowed. (not R0...R999) or a pointer register contains an unacceptable value.';

	16705:
		F_ADSErrorCodeExt := 'Unacceptable G-function index. (not 0...159) during execution.';

	16706:
		F_ADSErrorCodeExt := 'Unacceptable M-function index. (not 0...159) during execution.';

	16707:
		F_ADSErrorCodeExt := 'Unacceptable extended address. (not 1...9) during execution.';

	16708:
		F_ADSErrorCodeExt := 'Unacceptable index to the internal H-function.';

	16709:
		F_ADSErrorCodeExt := 'Machine data value unacceptable. (MDB) (not 0…7).';

	16720:
		F_ADSErrorCodeExt := 'Unacceptable change of parameters for the tool compensation during execution.';

	16721:
		F_ADSErrorCodeExt := 'Cannot calculate tool compensation.';

	16722:
		F_ADSErrorCodeExt := 'Tool compensation: The plane for the tool compensation cannot be changed here. This error occurred for instance by changing the tool plane when the compensation is turned on or active.';

	16723:
		F_ADSErrorCodeExt := 'Tool compensation: The D-Word is missing or invalid by turning on the tool compensation.';

	16724:
		F_ADSErrorCodeExt := 'Tool compensation: The specified tool radius is invalid because the value is less or equal zero.';

	16725:
		F_ADSErrorCodeExt := 'Tool compensation: The tool radius cannot be changed here';

	16726:
		F_ADSErrorCodeExt := 'Tool compensation: Collision Detection Table is full.';

	16727:
		F_ADSErrorCodeExt := 'Tool compensation: Internal error while turning on the contour collision detection.';

	16728:
		F_ADSErrorCodeExt := 'Tool compensation: Internal error within the contour collision detection: update reversed geo failed.';

	16729:
		F_ADSErrorCodeExt := 'Tool compensation: Unexpected combination of geometry types by active contour collision detection.';

	16730:
		F_ADSErrorCodeExt := 'Tool compensation: Programmed inner circle is smaller than the cutter radius';

	16731:
		F_ADSErrorCodeExt := 'Tool compensation: Bottle neck detection recognized contour violation';

	16732:
		F_ADSErrorCodeExt := 'Table for corrected entries is full';

	16733:
		F_ADSErrorCodeExt := 'Input table for tangential following is full';

	16734:
		F_ADSErrorCodeExt := 'Executing table for tangential following is full';

	16735:
		F_ADSErrorCodeExt := 'Geometric entry for tangential following cannot be calculated';

	16736:
		F_ADSErrorCodeExt := 'reserved';

	16737:
		F_ADSErrorCodeExt := 'reserved';

	16738:
		F_ADSErrorCodeExt := 'The actual active interpolation rules (g-code), zero-shifts, or rotation cannot be detected';

	16752:
		F_ADSErrorCodeExt := 'The NC has found an invalid parameter while loading an NC program.';

	16753:
		F_ADSErrorCodeExt := 'Invalid contour start position.';

	16754:
		F_ADSErrorCodeExt := 'Invalid internal entry index during execution of the retrace function.';

	16755:
		F_ADSErrorCodeExt := 'Invalid default G Code. False expression/syntax in default G Code.';

	16756:
		F_ADSErrorCodeExt := 'Error while opening the default G code file.';

		// NC - Group Error Codes 

	// 16896 - 17151
	16896:
		F_ADSErrorCodeExt := 'Group ID not allowed. e.g. because it has already been assigned, is less than OR equal TO zero, OR is greater than 255. Value range: [1 ... 255]';

	16897:
		F_ADSErrorCodeExt := 'Group type not allowed.';

	16898:
		F_ADSErrorCodeExt := 'Master axis index not allowed. Value range: 0-2';

	16899:
		F_ADSErrorCodeExt := 'Slave axis index not allowed. Value range: 0-7';

	16900:
		F_ADSErrorCodeExt := 'Internal Error. Possible causes: Not enough TC router memory, internal structures and pointers are erronouos or missing, check logger';

	16901:
		F_ADSErrorCodeExt := 'Invalid cycle time for statement execution task (SAF). Value range: 0.001-0.1';

	16902:
		F_ADSErrorCodeExt := 'GROUPERR_RANGE_MAXELEMENTSINAXIS.';

	16903:
		F_ADSErrorCodeExt := 'Invalid cycle time for the statement preparation task (SVB). Value range: 0.001-1.0';

	16904:
		F_ADSErrorCodeExt := 'Single step mode not allowed.';

	16905:
		F_ADSErrorCodeExt := 'Group deactivation not allowed.';

	16906:
		F_ADSErrorCodeExt := 'Statement execution state (SAF state) not allowed. Value range: 0-5';

	16907:
		F_ADSErrorCodeExt := 'The group does not have a channel, or the channel address has not been initialized.';

	16908:
		F_ADSErrorCodeExt := 'The group does not have a master axis (or axes) or the axis address(es) has (have) not been initialized.';

	16909:
		F_ADSErrorCodeExt := 'A new master/slave coupling is to be inserted into the group, but there is no valid address for the leading master axis.';

	16910:
		F_ADSErrorCodeExt := 'A master/slave coupling is to be inserted into the group, but there is no valid address for the slave axis.';

	16911:
		F_ADSErrorCodeExt := 'A master/slave coupling is to be inserted into the group, but there is no valid address for the slave set value generator.';

	16912:
		F_ADSErrorCodeExt := 'An axis in the group does not have an encoder, or the encoder address has not been initialized.';

	16913:
		F_ADSErrorCodeExt := 'An axis in the group does not have a controller, or the controller address has not been initialized.';

	16914:
		F_ADSErrorCodeExt := 'An axis in the group does not have a drive, or the drive address has not been initialized.';

	16915:
		F_ADSErrorCodeExt := 'A group (e.g. FIFO group) does not own a master setpoint generator or a setpoint generator address has not been initialized. Possibly, there may not be enough memory available.';

	16916:
		F_ADSErrorCodeExt := 'Group/axis does not have an axis interface from the NC to the PLC, or the axis interface address has not been initialized.';

	16917:
		F_ADSErrorCodeExt := 'An existing master/slave coupling is to be removed from the group, but there is no valid address for the slave axis.';

	16918:
		F_ADSErrorCodeExt := 'Table address unknown.';

	16919:
		F_ADSErrorCodeExt := 'The NcControl address has not been initialized.';

	16920:
		F_ADSErrorCodeExt := 'Axis is blocked for commands while persistent NC data are queued.';

	16921:
		F_ADSErrorCodeExt := 'The scaling mode MASTER-AUTOOFFSET is invalid because no reference table was found.';

	16922:
		F_ADSErrorCodeExt := 'The master axis start position does not permit synchronization.';

	16923:
		F_ADSErrorCodeExt := 'Slave coupling factor (gearing factor) of 0.0 is not allowed';

	16924:
		F_ADSErrorCodeExt := 'Insertion of master axis into group not allowed';

	16925:
		F_ADSErrorCodeExt := 'Deletion of master axis from group not allowed.';

	16926:
		F_ADSErrorCodeExt := 'Function/feature is not supported from the setpoint generator.';

	16927:
		F_ADSErrorCodeExt := 'Group has not been initialized. Although the group has been created, the rest of the initialization has not been performed.';

	16928:
		F_ADSErrorCodeExt := 'Group not ready / group not ready for new task';

	16929:
		F_ADSErrorCodeExt := 'Requested set velocity is not allowed';

	16930:
		F_ADSErrorCodeExt := 'Requested target position is not allowed (master axis)';

	16931:
		F_ADSErrorCodeExt := 'No enable for controller and/or feed (Master axis).';

	16932:
		F_ADSErrorCodeExt := 'Movement smaller than one encoder increment';

	16933:
		F_ADSErrorCodeExt := 'Drive not ready during axis start';

	16934:
		F_ADSErrorCodeExt := 'Invalid parameters of the emergency stop.';

	16935:
		F_ADSErrorCodeExt := 'The setpoint generator is inactive such that no instructions are accepted.';

	16936:
		F_ADSErrorCodeExt := 'Requested traverse distance is not allowed.';

	16937:
		F_ADSErrorCodeExt := 'Requested target position is not allowed (slave axis)';

	16938:
		F_ADSErrorCodeExt := 'No enable for controller and/or feed (slave axis)';

	16939:
		F_ADSErrorCodeExt := 'The activation position (position threshold) is out of range of the actual positioning';

	16940:
		F_ADSErrorCodeExt := 'The start or activation data of the external setpoint generation are not valid';

	16941:
		F_ADSErrorCodeExt := 'For changing the dynamic parameter (accel and decel), velocity must be in constant state';

	16942:
		F_ADSErrorCodeExt := 'Jerk less than or equal to 0.0 is not allowed.';

	16943:
		F_ADSErrorCodeExt := 'Acceleration less than or equal to 0.0 is not allowed';

	16944:
		F_ADSErrorCodeExt := 'Absolute deceleration value less than or equal to 0.0 is not allowed';

	16945:
		F_ADSErrorCodeExt := 'Set velocity less than or equal to 0.0 is not allowed';

	16946:
		F_ADSErrorCodeExt := 'Loss of precision when trying a positioning.';

	16947:
		F_ADSErrorCodeExt := 'Cycle time less than or equal to 0.0 is not allowed';

	16948:
		F_ADSErrorCodeExt := 'PTP data type <intasdouble> range exceeded. Loss of precision';

	16949:
		F_ADSErrorCodeExt := 'PTP LHL velocity profile cannot be generated. (Low-High-Low)';

	16950:
		F_ADSErrorCodeExt := 'PTP HML velocity profile cannot be generated. (High-Middle-Low).';

	16951:
		F_ADSErrorCodeExt := 'Start data address is invalid.';

	16952:
		F_ADSErrorCodeExt := 'Velocity override (start override) is not allowed';

	16953:
		F_ADSErrorCodeExt := 'Start type not allowed.';

	16954:
		F_ADSErrorCodeExt := 'Velocity overflow (overshoot in the velocity). Parameterized jerk is too weak.';

	16955:
		F_ADSErrorCodeExt := 'Start parameter for the axis structure is invalid.';

	16956:
		F_ADSErrorCodeExt := 'Override generator initialization parameter invalid.';

	16957:
		F_ADSErrorCodeExt := 'Slave axis has not set value generator';

	16958:
		F_ADSErrorCodeExt := 'Table is empty. Either the SVB table or the SAF table does not contain any entries.';

	16959:
		F_ADSErrorCodeExt := 'Table is full. The SVB table or the SAF table has no more free lines.';

	16960:
		F_ADSErrorCodeExt := 'No memory available. SVB memory allocation for dynamic entry in SAF table failed.';

	16961:
		F_ADSErrorCodeExt := 'Table already contains an entry.';

	16962:
		F_ADSErrorCodeExt := 'Stop is already active.';

	16963:
		F_ADSErrorCodeExt := 'Compensation has not been carried out over the full compensation section';

	16964:
		F_ADSErrorCodeExt := 'Internal parameters for the compensation are invalid.';

	16965:
		F_ADSErrorCodeExt := 'Start of compensation refused, because compensation is already active.';

	16966:
		F_ADSErrorCodeExt := 'Stop of compensation refused, because compensation is not active.';

	16967:
		F_ADSErrorCodeExt := 'Compensation type invalid.';

	16968:
		F_ADSErrorCodeExt := 'Axis address for compensation invalid.';

	16969:
		F_ADSErrorCodeExt := 'The slave address given for on-line coupling/decoupling is invalid.';

	16970:
		F_ADSErrorCodeExt := 'Coupling velocity invalid.';

	16971:
		F_ADSErrorCodeExt := 'The velocity of what is to become the master axis and the velocity of what is to become the slave axis are not constant, so that on-line coupling is not possible.';

	16972:
		F_ADSErrorCodeExt := 'Cycle time less than or equal to 0.0 is not allowed';

	16973:
		F_ADSErrorCodeExt := 'Decoupling task not allowed.';

	16974:
		F_ADSErrorCodeExt := 'The function cannot logically be executed, e.g. some commands are not possible and not allowed for slave axes.';

	16975:
		F_ADSErrorCodeExt := 'No valid table weighting has been set.';

	16976:
		F_ADSErrorCodeExt := 'Axis type, actual position type or end position type is not allowed.';

	16977:
		F_ADSErrorCodeExt := 'Function not presently supported.';

	16978:
		F_ADSErrorCodeExt := 'State of state machine invalid.';

	16979:
		F_ADSErrorCodeExt := 'Reference cam became free too soon';

	16980:
		F_ADSErrorCodeExt := 'Clearance monitoring between activation of the hardware latch and appearance of the sync pulse';

	16981:
		F_ADSErrorCodeExt := 'No memory available. The dynamic memory allocation for the set value generator, the SVB table or the SAF table has failed.';

	16982:
		F_ADSErrorCodeExt := 'The table slave axis has no active table.';

	16983:
		F_ADSErrorCodeExt := 'Function not allowed.';

	16984:
		F_ADSErrorCodeExt := 'Stopping compensation not allowed.';

	16985:
		F_ADSErrorCodeExt := 'The slave table cannot be activated, because it is currently being used.';

	16986:
		F_ADSErrorCodeExt := 'Master or slave axis is processing a job (e.g. positioning command) while coupling is requested';

	16987:
		F_ADSErrorCodeExt := 'Slave (start) parameter is incorrect.';

	16988:
		F_ADSErrorCodeExt := 'Slave type is incorrect. The slave type does not match up to the (SVB) start type.';

	16989:
		F_ADSErrorCodeExt := 'Axis stop is already active.';

	16990:
		F_ADSErrorCodeExt := 'Maximum number of tables per slavegenerator reached.';

	16991:
		F_ADSErrorCodeExt := 'The scaling mode is invalid.';

	16992:
		F_ADSErrorCodeExt := 'Controller enable for the axis or for a coupled slave axis is not present.';

	16993:
		F_ADSErrorCodeExt := 'Table not found.';

	16994:
		F_ADSErrorCodeExt := 'Incorrect table type.';

	16995:
		F_ADSErrorCodeExt := 'Single step mode is still being processed for a group or axis and a new task was requested.';

	16996:
		F_ADSErrorCodeExt := 'Group task unknown (asynchronous table entry).';

	16997:
		F_ADSErrorCodeExt := 'Group function unknown (synchronous function)';

	16998:
		F_ADSErrorCodeExt := 'Group task for slave not allowed';

	16999:
		F_ADSErrorCodeExt := 'Group function for slave not allowed';

	17000:
		F_ADSErrorCodeExt := 'NCI Setpoint Generator is Inactive';

	17001:
		F_ADSErrorCodeExt := 'Startposition=Setpoint Position. Invalid position parameters.';

	17002:
		F_ADSErrorCodeExt := 'Parameters of the delay-generator are invalid.';

	17003:
		F_ADSErrorCodeExt := 'External parameters of the superimposed instruction are invalid.';

	17004:
		F_ADSErrorCodeExt := 'Invalid override type.';

	17005:
		F_ADSErrorCodeExt := 'Activation position under/overrun. (e.g. when exchanging a cam table).';

	17006:
		F_ADSErrorCodeExt := 'Activation impossible: Master is not moving.';

	17007:
		F_ADSErrorCodeExt := 'Activation mode not possible. Slave axis is moving.';

	17008:
		F_ADSErrorCodeExt := 'Start parameter for the compensation is invalid. Acceleration (>0) Deceleration (>0) Process velocity (>0)';

	17009:
		F_ADSErrorCodeExt := 'Start parameter for the compensation is invalid. Velocity camber is negative.';

	17010:
		F_ADSErrorCodeExt := 'Start parameter for the compensation is invalid. The section on which the compensation is to occur is not positive.';

	17011:
		F_ADSErrorCodeExt := 'Target position under/overrun.';

	17012:
		F_ADSErrorCodeExt := 'Target position will be under/overrun.';

	17013:
		F_ADSErrorCodeExt := 'Group Parameter is Invalid';

	17014:
		F_ADSErrorCodeExt := 'Joint Error at Start of Setpoint Generation';

	17015:
		F_ADSErrorCodeExt := 'Dynamic parameters not permitted.';

	17017:
		F_ADSErrorCodeExt := 'The New Target Position is Invalid or Cannot be Reached';

	17018:
		F_ADSErrorCodeExt := 'New Velocity for Moving or the Final Target Velocity is Invalid';

	17019:
		F_ADSErrorCodeExt := 'The Final Velocity or the New Target Position is Invalid';

	17020:
		F_ADSErrorCodeExt := 'The New Moving Velocity is Invalid';

	17021:
		F_ADSErrorCodeExt := 'Internal Starting Mode is Invalid';

	17022:
		F_ADSErrorCodeExt := 'A requested motion command could not be realized (BISECTION)';

	17023:
		F_ADSErrorCodeExt := 'The new target position either has been overrun or will be overrun.';

	17024:
		F_ADSErrorCodeExt := 'Group not ready / group not ready for new task';

	17025:
		F_ADSErrorCodeExt := 'The parameters of the oriented stop (O-Stop) are not admitted. The modulo-target position should not be smaller than zero and not larger or equal than the encoder mod-period.';

	17026:
		F_ADSErrorCodeExt := 'The modulo target position of the modulo-start is invalid';

	17027:
		F_ADSErrorCodeExt := 'The online change activation mode is invalid';

	17028:
		F_ADSErrorCodeExt := 'The parameterized jerk rate is smaller than the minimum jerk rate.';

	17029:
		F_ADSErrorCodeExt := 'The parameterized acceleration or deceleration is not permitted';

	17030:
		F_ADSErrorCodeExt := 'The parameterized velocity is not permitted. Less than 0';

	17031:
		F_ADSErrorCodeExt := 'A activation cannot be executed due to a pending activation';

	17032:
		F_ADSErrorCodeExt := 'Illegal combination of different cycle times within an axis group';

	17033:
		F_ADSErrorCodeExt := 'Illegal motion reversal. The previous system state is restored.';

	17034:
		F_ADSErrorCodeExt := 'Illegal moment for an axis command because there is an old axis command with activation position still active';

	17035:
		F_ADSErrorCodeExt := 'Error in the stop-calculation routine. The previous system state is restored.';

	17036:
		F_ADSErrorCodeExt := 'A command with activation position cannot fully be performed because the remaining path is too short';

	17037:
		F_ADSErrorCodeExt := 'Illegal decouple type when decoupling a slave axis.';

	17038:
		F_ADSErrorCodeExt := 'Illegal target velocity when decoupling a slave axis.';

	17039:
		F_ADSErrorCodeExt := 'The command new dynamic parameter cannot be performed since this would require a new target velocity';

	17040:
		F_ADSErrorCodeExt := 'A command with activation position cannot be performed because the axis is already in the brake phase';

	17041:
		F_ADSErrorCodeExt := 'Decouple routine of slave axis does not return a valid solution';

	17042:
		F_ADSErrorCodeExt := 'Command cannot be executed because the command buffer is full filled.';

	17043:
		F_ADSErrorCodeExt := 'Command is rejected due to an internal error in the Look Ahead.';

	17044:
		F_ADSErrorCodeExt := 'Command is rejected because the segment target velocity is not realized.';

	17045:
		F_ADSErrorCodeExt := 'Successive commands have the same final position. So the moving distance is zero.';

	17046:
		F_ADSErrorCodeExt := 'Logical positioning direction is inconsistent with the direction of the buffer command';

	17047:
		F_ADSErrorCodeExt := 'Command is rejected because the remaining positioning length is to small.';

	17050:
		F_ADSErrorCodeExt := 'Restart has Failed. There is already a motion command within the PTP buffer.';

	17051:
		F_ADSErrorCodeExt := 'Collection error for invalid start parameters. Base frequency < 0, StartFreq <1, StepCount <1 or StepCount >200, BaseAmpl <=0, StepDuration <=0, StopFreq >=1/(2*CycleTime)';

	17052:
		F_ADSErrorCodeExt := 'Reference cam is not found.';

	17053:
		F_ADSErrorCodeExt := 'Reference cam became not free';

	17054:
		F_ADSErrorCodeExt := 'IO sync pulse was not found (only when using hardware latch)';

	17055:
		F_ADSErrorCodeExt := 'The Used Buffer Mode is Unknown or not Supported in this Context';

	17056:
		F_ADSErrorCodeExt := 'Group/axis consequential error. Resulting from another causative error related to another axis within the group.';

	17057:
		F_ADSErrorCodeExt := 'Velocity reduction factor for C0/C1 transition is not allowed';

	17058:
		F_ADSErrorCodeExt := 'Critical angle at segment transition not allowed.';

	17059:
		F_ADSErrorCodeExt := 'Radius of the tolerance sphere is in an invalid range';

	17060:
		F_ADSErrorCodeExt := 'Not implemented.';

	17061:
		F_ADSErrorCodeExt := 'Start type error.';

	17062:
		F_ADSErrorCodeExt := 'Not implemented.';

	17063:
		F_ADSErrorCodeExt := 'Blending with given parameters not possible';

	17064:
		F_ADSErrorCodeExt := 'Not implemented.';

	17065:
		F_ADSErrorCodeExt := 'Curve velocity reduction method not allowed.';

	17066:
		F_ADSErrorCodeExt := 'Minimum velocity is less than 0.';

	17067:
		F_ADSErrorCodeExt := 'Power function input not allowed.';

	17068:
		F_ADSErrorCodeExt := 'Dynamic change parameter not allowed.';

	17069:
		F_ADSErrorCodeExt := 'Memory allocation error.';

	17070:
		F_ADSErrorCodeExt := 'The calculated end position differs from the end position in the nc instruction (internal error).';

	17071:
		F_ADSErrorCodeExt := 'Calculate remaining chord length is invalid.';

	17072:
		F_ADSErrorCodeExt := 'Starting the set value generator (SVB, SAF) has been refused, since the SVB task is already active.';

	17073:
		F_ADSErrorCodeExt := 'SVB parameter not allowed. Set value generator (SVB) results in logical error.';

	17074:
		F_ADSErrorCodeExt := 'Velocity reduction factor not allowed. Parameter that controls reduction of the velocity at segment transition is invalid.';

	17075:
		F_ADSErrorCodeExt := 'The helix has degenerated to a circle, and should be entered as such.';

	17076:
		F_ADSErrorCodeExt := 'The helix has degenerated to a straight line, and should be entered as such.';

	17077:
		F_ADSErrorCodeExt := 'Guider parameter not allowed.';

	17078:
		F_ADSErrorCodeExt := 'Invalid segment address. Invalid geometry or does not have a valid dynamic structure address.';

	17079:
		F_ADSErrorCodeExt := 'Unparameterized generator. The SVB generator is not yet parameterized and is therefore unable to operate.';

	17080:
		F_ADSErrorCodeExt := 'Unparameterized table. The table has no information concerning the address of the corresponding dynamic generator.';

	17082:
		F_ADSErrorCodeExt := 'The calculation of the arc length of the smoothed path failed (internal error).';

	17083:
		F_ADSErrorCodeExt := 'The radius of the tolerance ball is too small (smaller than 0.1 mm).';

	17084:
		F_ADSErrorCodeExt := 'Error while calculating DXD-Software-Limit switches (internal error)';

	17085:
		F_ADSErrorCodeExt := 'NC-Block violates software limit switches of the group. Therefore the geometric entry is denied with an error.';

	17086:
		F_ADSErrorCodeExt := 'Internal error in the evaluation of a possible software limit switch violation for the segment with the block-number xx.';

	17087:
		F_ADSErrorCodeExt := 'Invalid reference speed type.';

	17088:
		F_ADSErrorCodeExt := 'Interpolating group contains axes of an incorrect axis type. An interpolating 3D group may only contain continuously guided axes of axis type 1 (SERVO).';

	17089:
		F_ADSErrorCodeExt := 'Scalar product cannot be calculated. The length of one of the given vectors is 0.0.';

	17090:
		F_ADSErrorCodeExt := 'Inverse cosine cannot be calculated. The length of one of the given vectors is 0.0.';

	17091:
		F_ADSErrorCodeExt := 'Invalid table entry type. The given table entry type is unknown.';

	17092:
		F_ADSErrorCodeExt := 'Invalid DIN66025 information type. (INTERNAL ERROR) The given DIN66025 information type is unknown. Known types: G0, G1, G2, G3, G17, G18, G19.';

	17093:
		F_ADSErrorCodeExt := 'Invalid dimension. (INTERNAL ERROR) The CNC dimension is unknown.';

	17094:
		F_ADSErrorCodeExt := 'Geometrical object is not a straight line. The given object, interpreted as a straight line, has a length of 0.0.';

	17095:
		F_ADSErrorCodeExt := 'Geometrical object is not a circle. Interpreted as a circular arc, the given object has a length of 0.0, or an angle of 0.0 or a radius of 0.0.';

	17096:
		F_ADSErrorCodeExt := 'Geometrical object is not a helix. Interpreted as a circular arc, the given object has a length of 0.0, or an angle of 0.0, or a radius of 0.0. or a height of 0.0.';

	17097:
		F_ADSErrorCodeExt := 'Set velocity less than or equal to 0.0 is invalid.';

	17098:
		F_ADSErrorCodeExt := 'The address supplied for the look-ahead is invalid.';

	17099:
		F_ADSErrorCodeExt := 'Starting the set value generator (SAF) has been refused, since the SAF task is already active.';

	17100:
		F_ADSErrorCodeExt := 'CNC set value generation not active. Stop or change of override refused, because the set value generation is not active.';

	17101:
		F_ADSErrorCodeExt := 'CNC set value generation in the stop phase. Stop or change of override refused, because the set value generation is in the stop phase.';

	17102:
		F_ADSErrorCodeExt := 'Override not allowed. An override of less than 0.0 % or more than 100.0 % is invalid.';

	17103:
		F_ADSErrorCodeExt := 'The table address given for the initialization of the set value generator is invalid, or no valid logger connection (report file) is present.';

	17104:
		F_ADSErrorCodeExt := 'Invalid table entry type. The given table entry type is unknown.';

	17105:
		F_ADSErrorCodeExt := 'Memory allocation for the table has failed.';

	17106:
		F_ADSErrorCodeExt := 'Memory allocation for the filter has failed.';

	17107:
		F_ADSErrorCodeExt := 'Filter parameter is not allowed.';

	17108:
		F_ADSErrorCodeExt := 'Delete Distance to go (only interpolation) failed. This error occurred, if e.g. the command DelDTG was not programmed in the actual movement of the nc program.';

	17109:
		F_ADSErrorCodeExt := 'The setpoint generator of the flying saw generates incompatible values (internal error).';

	17110:
		F_ADSErrorCodeExt := 'Axis will be stopped since otherwise it will overrun its target position (old PTP setpoint generator)';

	17111:
		F_ADSErrorCodeExt := 'Internal error in the transformation from slave to master.';

	17112:
		F_ADSErrorCodeExt := 'Wrong direction in the transformation of slave to master.';

	17114:
		F_ADSErrorCodeExt := 'Parameter of Motion Function (MF) table incorrect. This may refer to the first time created data set or to online changed data.';

	17115:
		F_ADSErrorCodeExt := 'Parameter of Motion Function (MF) table incorrect. The error cause can be, that an active MF point (no IGNORE point) points at a passive MF point (IGNORE point).';

	17116:
		F_ADSErrorCodeExt := 'Internal error by using Motion Function (MF). This error cannot be solved by the user. Please ask the TwinCAT Support.';

	17117:
		F_ADSErrorCodeExt := 'Axis coupling with synchronization generator declined because of incorrect axis dynamic values';

	17118:
		F_ADSErrorCodeExt := 'Coupling conditions of synchronization generator incorrect';

	17119:
		F_ADSErrorCodeExt := 'Moving profile of synchronization generator declines dynamic limit of slave axis or required characteristic of profile';

	17120:
		F_ADSErrorCodeExt := 'The encoder generator parameter is not allowed.';

	17121:
		F_ADSErrorCodeExt := 'The external (Fifo) generator parameter is not allowed.';

	17122:
		F_ADSErrorCodeExt := 'The external generator cannot be started, as it is already active.';

	17123:
		F_ADSErrorCodeExt := 'The external generator cannot be stopped, as it is not active.';

	17124:
		F_ADSErrorCodeExt := 'NC-Block with auxiliary axis violates software limit switches of the group.';

	17125:
		F_ADSErrorCodeExt := 'NC-Block type Bezier spline curve contains a cusp (singularity). The Bezier spline curve contain a cusp.';

	17127:
		F_ADSErrorCodeExt := 'Value FOR dead TIME compensation NOT allowed.';

	17128:
		F_ADSErrorCodeExt := 'GROUPERR_RANGE_NOMOTIONWINDOW';

	17129:
		F_ADSErrorCodeExt := 'GROUPERR_RANGE_NOMOTIONFILTERTIME';

	17130:
		F_ADSErrorCodeExt := 'GROUPERR_RANGE_TIMEUNITFIFO';

	17131:
		F_ADSErrorCodeExt := 'GROUPERR_RANGE_OVERRIDETYPE';

	17132:
		F_ADSErrorCodeExt := 'GROUPERR_RANGE_OVERRIDECHANGETIME';

	17133:
		F_ADSErrorCodeExt := 'GROUPERR_FIFO_INVALIDDIMENSION';

	17134:
		F_ADSErrorCodeExt := 'GROUPERR_ADDR_FIFOTABLE';

	17135:
		F_ADSErrorCodeExt := 'Axis is locked for motion commands because a stop command is still active.';

	17136:
		F_ADSErrorCodeExt := 'Invalid number of auxiliary axes.';

	17137:
		F_ADSErrorCodeExt := 'The velocity reduction parameters FOR the auxiliary axes are inconsistent.';

	17138:
		F_ADSErrorCodeExt := 'The dynamic parameters FOR the auxiliary axes are inconsistent.';

	17139:
		F_ADSErrorCodeExt := 'The coupling parameters FOR the auxiliary axes are inconsistent.';

	17140:
		F_ADSErrorCodeExt := 'The auxiliary axis entry is empty (no axis motion).';

	17142:
		F_ADSErrorCodeExt := 'The LIMIT FOR velocity reduction OF the auxiliary axes is invalid.';

	17144:
		F_ADSErrorCodeExt := 'Block search - segment NOT found. The segment specified as a parameter could not be found by the end of the NC program.';

	17145:
		F_ADSErrorCodeExt := 'Blocksearch – invalid remaining segment length. The remaining travel in the parameter fLength is incorrectly parameterized.';

	17147:
		F_ADSErrorCodeExt := 'INTERNAL Error in the Context OF Coupled Axes (Slave Axes).';

	17148:
		F_ADSErrorCodeExt := 'Parameter FOR the Maximum Number OF Jobs (Entries) TO be Transferred is Invalid';

	17151:
		F_ADSErrorCodeExt := 'Customer Specific Error';

		// NC - Axis Error Codes (Includes TF5055 Flying Saw)

	// 17152 - 17312)
	17152:
		F_ADSErrorCodeExt := 'Axis ID not allowed.';

	17153:
		F_ADSErrorCodeExt := 'Axis type not allowed.';

	17158:
		F_ADSErrorCodeExt := 'Slow manual velocity not allowed.';

	17159:
		F_ADSErrorCodeExt := 'Fast manual velocity not allowed.';

	17160:
		F_ADSErrorCodeExt := 'High speed not allowed.';

	17161:
		F_ADSErrorCodeExt := 'Acceleration not allowed.';

	17162:
		F_ADSErrorCodeExt := 'Deceleration not allowed.';

	17163:
		F_ADSErrorCodeExt := 'Jerk not allowed.';

	17164:
		F_ADSErrorCodeExt := 'Delay time between position and velocity is not allowed (dead time compensation).';

	17165:
		F_ADSErrorCodeExt := 'Override type not allowed.';

	17166:
		F_ADSErrorCodeExt := 'NCI: Velo-Jump-Factor not allowed.';

	17167:
		F_ADSErrorCodeExt := 'NCI: Size of tolerance sphere for auxiliary axis invalid.';

	17168:
		F_ADSErrorCodeExt := 'NCI: Value for maximum deviation for auxiliary axis invalid.';

	17170:
		F_ADSErrorCodeExt := 'Referencing velocity in direction of cam not allowed.';

	17171:
		F_ADSErrorCodeExt := 'Referencing velocity in sync direction not allowed.';

	17172:
		F_ADSErrorCodeExt := 'Pulse width in positive direction not allowed';

	17173:
		F_ADSErrorCodeExt := 'Pulse width in negative direction not allowed';

	17174:
		F_ADSErrorCodeExt := 'The value for the pulse width in positive direction is not allowed (pulsed operation).';

	17175:
		F_ADSErrorCodeExt := 'The value for the pulse width in negative direction is not allowed (pulsed operation).';

	17176:
		F_ADSErrorCodeExt := 'The value for the creep distance in positive direction is not allowed.';

	17177:
		F_ADSErrorCodeExt := 'The value for the creep distance in negative direction is not allowed.';

	17178:
		F_ADSErrorCodeExt := 'The value for the braking distance in positive direction is not allowed.';

	17179:
		F_ADSErrorCodeExt := 'The value for the braking distance in negative direction is not allowed.';

	17180:
		F_ADSErrorCodeExt := 'The value for the braking time in positive direction is not allowed.';

	17181:
		F_ADSErrorCodeExt := 'The value for the braking time in negative direction is not allowed.';

	17182:
		F_ADSErrorCodeExt := 'The value for the switching time from high to low speed is not allowed.';

	17183:
		F_ADSErrorCodeExt := 'The value for the creep distance for an explicit stop is not allowed.';

	17184:
		F_ADSErrorCodeExt := 'The value for the motion monitoring time is not allowed.';

	17185:
		F_ADSErrorCodeExt := 'The value for the activation of the position window monitoring is not allowed.';

	17186:
		F_ADSErrorCodeExt := 'The value for the activation of target window monitoring is not allowed.';

	17187:
		F_ADSErrorCodeExt := 'The value for the activation of loop movement is not allowed.';

	17188:
		F_ADSErrorCodeExt := 'The value for the motion monitoring time is not allowed.';

	17189:
		F_ADSErrorCodeExt := 'The value for the target window is not allowed.';

	17190:
		F_ADSErrorCodeExt := 'The value for the position window is not allowed.';

	17191:
		F_ADSErrorCodeExt := 'The value for the position window monitoring time is not allowed.';

	17192:
		F_ADSErrorCodeExt := 'The value for the loop movement is not allowed.';

	17193:
		F_ADSErrorCodeExt := 'The value for the axis cycle time is not allowed.';

	17194:
		F_ADSErrorCodeExt := 'The value for the stepper motor operating mode is not allowed.';

	17195:
		F_ADSErrorCodeExt := 'The value for the displacement associated with one step of the stepper motor is not allowed (step scaling).';

	17196:
		F_ADSErrorCodeExt := 'The value for the minimum speed of the stepper motor speed profile is not allowed.';

	17197:
		F_ADSErrorCodeExt := 'The value for the number of steps per speed level of the setpoint generation is not allowed.';

	17198:
		F_ADSErrorCodeExt := 'The value containing the flags for the interpretation of position and velocity units is not allowed.';

	17199:
		F_ADSErrorCodeExt := 'The value for the maximum permitted velocity is not allowed.';

	17200:
		F_ADSErrorCodeExt := 'The value for the motion monitoring window is not allowed.';

	17201:
		F_ADSErrorCodeExt := 'The value for the activation of the PEH time monitoring is not allowed (PEH: positioning end and halt).';

	17202:
		F_ADSErrorCodeExt := 'The value for the PEH monitoring time (timeout) is not allowed (PEH: positioning end and halt). Default value: 5s';

	17203:
		F_ADSErrorCodeExt := 'Parameter "Brake Release Delay" is invalid';

	17204:
		F_ADSErrorCodeExt := 'Parameter "NC Data Persistence" is invalid';

	17205:
		F_ADSErrorCodeExt := 'Parameter for Error Reaction Mode is invalid';

	17206:
		F_ADSErrorCodeExt := 'Parameter for the Error Reaction Delay is invalid';

	17207:
		F_ADSErrorCodeExt := 'Parameter "Use actual values in deactivated state" is invalid';

	17208:
		F_ADSErrorCodeExt := 'Parameter "Allow Motion Commands for Slave Axes" is invalid';

	17209:
		F_ADSErrorCodeExt := 'Parameter "Allow Motion Commands for axis in external setpoint generation" is invalid';

	17210:
		F_ADSErrorCodeExt := 'Parameter "Fading Acceleration" is invalid';

	17211:
		F_ADSErrorCodeExt := 'The value for the signal type of the Fast Axis Stop is not allowed [0...5].';

	17216:
		F_ADSErrorCodeExt := 'Axis has not been initialized.';

	17217:
		F_ADSErrorCodeExt := 'Axis does not have a group, or the group address has not been initialized (group contains the setpoint generation).';

	17218:
		F_ADSErrorCodeExt := 'The axis does not have an encoder, or the encoder address has not been initialized.';

	17219:
		F_ADSErrorCodeExt := 'An axis does not have a controller, or the controller address has not been initialized.';

	17220:
		F_ADSErrorCodeExt := 'The axis does not have a drive, or the drive address has not been initialized.';

	17221:
		F_ADSErrorCodeExt := 'Axis does not have an axis interface from the PLC to the NC, or the axis interface address has not been initialized.';

	17222:
		F_ADSErrorCodeExt := 'Axis does not have an axis interface from the NC to the PLC, or the axis interface address has not been initialized.';

	17223:
		F_ADSErrorCodeExt := 'The size of the axis interface from the NC to the PLC (NC to PLC) is not allowed.';

	17224:
		F_ADSErrorCodeExt := 'The size of the axis interface from the PLC to the NC is not allowed.';

	17238:
		F_ADSErrorCodeExt := 'Controller enable for the axis is not present.';

	17239:
		F_ADSErrorCodeExt := 'Missing negative feed enable for negative motion direction.';

	17240:
		F_ADSErrorCodeExt := 'Missing positive feed enable for positive motion direction.';

	17241:
		F_ADSErrorCodeExt := 'Set velocity not allowed.';

	17242:
		F_ADSErrorCodeExt := 'Movement smaller than one encoder increment not allowed';

	17243:
		F_ADSErrorCodeExt := 'The set acceleration has exceeded the maximum permitted acceleration or deceleration parameters of the axis';

	17244:
		F_ADSErrorCodeExt := 'The PEH time monitoring time that follows positioning has elapsed, the target position window has not been reached.';

	17245:
		F_ADSErrorCodeExt := 'The actual position of the axis has not changed or has changed only slightly during the motion monitoring time.';

	17246:
		F_ADSErrorCodeExt := 'Looping distance less than breaking distance.';

	17247:
		F_ADSErrorCodeExt := 'Starting velocity not allowed.';

	17248:
		F_ADSErrorCodeExt := 'Final velocity not allowed.';

	17249:
		F_ADSErrorCodeExt := 'Time range exceeded (future). The calculated position lies too far in the future.';

	17250:
		F_ADSErrorCodeExt := 'Time range exceeded (past)" The calculated position lies too far in the past.';

	17251:
		F_ADSErrorCodeExt := 'The requested position cannot be determined.';

	17252:
		F_ADSErrorCodeExt := 'Position indeterminable (conflicting direction of travel)';

	17264:
		F_ADSErrorCodeExt := 'No slave coupling possible (velocity violation)';

	17265:
		F_ADSErrorCodeExt := 'No slave coupling possible (acceleration violation)';

	17266:
		F_ADSErrorCodeExt := 'The synchronization profile would violate the lower end position of the slave.';

	17267:
		F_ADSErrorCodeExt := 'The synchronization profile would violate the upper end position of the slave.';

	17268:
		F_ADSErrorCodeExt := 'The synchronization profile would violate the user limit position Options.PositionLimitMin.';

	17269:
		F_ADSErrorCodeExt := 'The synchronization profile would violate the user limit position Options.PositionLimitMax.';

	17270:
		F_ADSErrorCodeExt := 'The synchronization point lies under the starting point. As a result, the profile swings under both the start position and the synchronous position.';

	17271:
		F_ADSErrorCodeExt := 'The synchronization profile would swing back under the slave start position of the flying saw.';

	17272:
		F_ADSErrorCodeExt := 'The synchronization point lies under the starting point. The synchronization profile would swing beyond the slave start position of the flying saw.';

	17273:
		F_ADSErrorCodeExt := 'The synchronization profile would swing beyond the slave synchronous position of the flying saw.';

	17274:
		F_ADSErrorCodeExt := 'The maximum velocity of the synchronization profile is higher than the maximum velocity of the slave axis.';

	17275:
		F_ADSErrorCodeExt := 'The maximum velocity of the synchronization profile is higher than the maximum velocity of the slave axis.';

	17276:
		F_ADSErrorCodeExt := 'The maximum velocity of the synchronization profile would be higher than the synchronous velocity.';

	17277:
		F_ADSErrorCodeExt := 'The maximum velocity of the synchronization profile would be higher than the starting velocity and synchronous velocity.';

	17278:
		F_ADSErrorCodeExt := 'The maximum velocity of the synchronization profile would be higher than the synchronous velocity.';

	17279:
		F_ADSErrorCodeExt := 'The maximum velocity of the synchronization profile would be higher than the starting velocity and synchronous velocity.';

	17280:
		F_ADSErrorCodeExt := 'The minimum velocity of the synchronization profile lies below the synchronous velocity.';

	17281:
		F_ADSErrorCodeExt := 'The minimum velocity of the synchronization profile lies below the starting velocity.';

	17282:
		F_ADSErrorCodeExt := 'The minimum velocity of the synchronization profile lies below the synchronous velocity.';

	17283:
		F_ADSErrorCodeExt := 'The minimum velocity of the synchronization profile lies below the starting velocity.';

	17286:
		F_ADSErrorCodeExt := 'The velocity of the flying saw swings below zero; the motion is reversed.';

	17287:
		F_ADSErrorCodeExt := 'The velocity of the flying saw swings below zero; the motion is reversed.';

	17288:
		F_ADSErrorCodeExt := 'The maximum acceleration of the synchronization profile would be higher than the maximum acceleration of the slave axis.';

	17289:
		F_ADSErrorCodeExt := 'The maximum deceleration of the synchronization profile would be higher than the maximum deceleration of the slave axis.';

	17290:
		F_ADSErrorCodeExt := 'The maximum jerk of the synchronization profile would be higher than the maximum jerk of the slave axis.';

	17291:
		F_ADSErrorCodeExt := 'The maximum jerk of the synchronization profile would be higher than the maximum jerk of the slave axis.';

	17312:
		F_ADSErrorCodeExt := 'Axis consequential error. Consequential error resulting from another causative error related to another axis.';

		// NC - Encoder Error Codes 

	// 17408 - 17571
	17408:
		F_ADSErrorCodeExt := 'Encoder ID NOT allowed';

	17409:
		F_ADSErrorCodeExt := 'Encoder type not allowed';

	17410:
		F_ADSErrorCodeExt := 'The value for the encoder (operating) mode is not allowed.';

	17411:
		F_ADSErrorCodeExt := 'Encoder counting direction inverted?';

	17412:
		F_ADSErrorCodeExt := 'The flag for the referencing status is not allowed.';

	17413:
		F_ADSErrorCodeExt := 'The value for the number of encoder increments for each physical rotation of the encoder is not allowed.';

	17414:
		F_ADSErrorCodeExt := 'The value for the scaling factor is not allowed.';

	17415:
		F_ADSErrorCodeExt := 'The value for the position offset of the encoder is not allowed.';

	17416:
		F_ADSErrorCodeExt := 'The value for the encoders modulo factor is not allowed.';

	17417:
		F_ADSErrorCodeExt := 'The value for the actual position filter time is not allowed (P-T1 filter).';

	17418:
		F_ADSErrorCodeExt := 'The value for the actual velocity filter time is not allowed (P-T1 filter).';

	17419:
		F_ADSErrorCodeExt := 'The value for the actual acceleration filter time is not allowed (P-T1 filter).';

	17420:
		F_ADSErrorCodeExt := 'The value of the SAF cycle time for the calculation of actual values is not allowed (e.g. is less than or equal to zero).';

	17421:
		F_ADSErrorCodeExt := 'Configuration of the selected units is invalid” E.g. settings for modulo position, velocity per minute etc. lead to an error.';

	17422:
		F_ADSErrorCodeExt := 'The value for the activation of the actual position correction ("measuring system error correction") is not allowed.';

	17423:
		F_ADSErrorCodeExt := 'The value for the actual position correction filter time is not allowed (P-T1 filter).';

	17424:
		F_ADSErrorCodeExt := 'Search direction for referencing cam inverted.';

	17425:
		F_ADSErrorCodeExt := 'Search direction for sync pulse (zero pulse) inverted.';

	17426:
		F_ADSErrorCodeExt := 'The value of the reference position in a referencing procedure is not allowed.';

	17427:
		F_ADSErrorCodeExt := 'Clearance monitoring between activation of the hardware latch and appearance of the sync pulse.';

	17428:
		F_ADSErrorCodeExt := 'Minimum clearance between activation of the hardware latch and appearance of the sync pulse.';

	17429:
		F_ADSErrorCodeExt := 'The value of the activation or deactivation of the external sync pulse in a referencing procedure is not allowed.';

	17430:
		F_ADSErrorCodeExt := 'Scaling of the noise rate on simulation encoder is not allowed.';

	17431:
		F_ADSErrorCodeExt := 'The value for the tolerance window for the modulo-axis-start is invalid.';

	17432:
		F_ADSErrorCodeExt := 'The value for the encoder reference mode is not allowed, resp. is not supported for this encoder type.';

	17433:
		F_ADSErrorCodeExt := 'The value for the encoder evaluation direction (log. counter direction) is not allowed.';

	17434:
		F_ADSErrorCodeExt := 'The value for the encoder reference system is invalid.';

	17435:
		F_ADSErrorCodeExt := 'When starting the TC system the value for the encoder position initialization mode is invalid.';

	17436:
		F_ADSErrorCodeExt := 'Encoder sign interpretation (UNSIGNED- / SIGNED- data type) is invalid.';

	17437:
		F_ADSErrorCodeExt := 'The value for the encoder homing sensor source is not allowed.';

	17440:
		F_ADSErrorCodeExt := 'Software minimum end location monitoring not allowed.';

	17441:
		F_ADSErrorCodeExt := 'Software maximum end location monitoring not allowed.';

	17442:
		F_ADSErrorCodeExt := 'Actual value setting is outside the value range.';

	17443:
		F_ADSErrorCodeExt := 'Software end location minimum not allowed.';

	17444:
		F_ADSErrorCodeExt := 'Software end location maximum not allowed.';

	17445:
		F_ADSErrorCodeExt := 'The value for the filter mask of the encoder raw data in increments is invalid.';

	17446:
		F_ADSErrorCodeExt := 'Reference mask for the raw data of the encoder is invalid';

	17447:
		F_ADSErrorCodeExt := 'Parameter Dead Time Compensation Mode (Encoder) is Invalid';

	17448:
		F_ADSErrorCodeExt := 'Parameter “Control Bits of Dead Time Compensation” (Encoder) is Invalid';

	17449:
		F_ADSErrorCodeExt := 'Parameter “Time Related Shift of Dead Time Compensation Mode” (Encoder) is Invalid';

	17456:
		F_ADSErrorCodeExt := 'Hardware latch activation (encoder), hardware latch was implicitly initated by the referencing procedure.';

	17457:
		F_ADSErrorCodeExt := 'External hardware latch activation (encoder) via ADS has already been activated, but no valid latch value present';

	17458:
		F_ADSErrorCodeExt := 'External hardware latch activation (encoder), hardware still signals a valid latch value.';

	17459:
		F_ADSErrorCodeExt := 'External hardware latch activation (encoder), hardware still signalling that the external latch value is still valid.';

	17460:
		F_ADSErrorCodeExt := 'An encoder function has been activated that is currently not released for use, or which is not even implemented.';

	17461:
		F_ADSErrorCodeExt := 'An encoder function can not been activated because this functionality is already active.';

	17472:
		F_ADSErrorCodeExt := 'Encoder has not been initialized.';

	17473:
		F_ADSErrorCodeExt := 'The encoder does not have an axis, or the axis address has not been initialized.';

	17474:
		F_ADSErrorCodeExt := 'The drive does not have a valid I/O input address in the process image.';

	17475:
		F_ADSErrorCodeExt := 'The encoder does not have a valid I/O output address in the process image.';

	17488:
		F_ADSErrorCodeExt := 'The encoders incremental counter has underflowed.';

	17489:
		F_ADSErrorCodeExt := 'The encoders incremental counter has overflowed.';

	17504:
		F_ADSErrorCodeExt := 'Minimum Software Position Limit (Axis Start).';

	17505:
		F_ADSErrorCodeExt := 'Maximum Software Position Limit (Axis Start).';

	17506:
		F_ADSErrorCodeExt := 'Minimum Software Position Limit (Positioning Process).';

	17507:
		F_ADSErrorCodeExt := 'Maximum Software Position Limit (Positioning Process).';

	17508:
		F_ADSErrorCodeExt := 'Encoder hardware error.';

	17509:
		F_ADSErrorCodeExt := 'Position initialization error at system start.';

	17510:
		F_ADSErrorCodeExt := 'Invalid IO data for more than n subsequent NC cycles (encoder)';

	17511:
		F_ADSErrorCodeExt := 'Invalid Actual Position (Encoder)';

	17512:
		F_ADSErrorCodeExt := 'Invalid IO Input Data (Error Type 1)';

	17513:
		F_ADSErrorCodeExt := 'Invalid IO Input Data (Error Type 2)';

	17520:
		F_ADSErrorCodeExt := 'SSI transformation fault or not finished.';

	17570:
		F_ADSErrorCodeExt := 'ENCERR_ADDR_CONTROLLER';

	17571:
		F_ADSErrorCodeExt := 'ENCERR_INVALID_CONTROLLERTYPE';

		// NC - Controller Error Codes 

	// 17664 - 17828
	17664:
		F_ADSErrorCodeExt := 'Controller ID not allowed.';

	17665:
		F_ADSErrorCodeExt := 'Controller type not allowed.';

	17666:
		F_ADSErrorCodeExt := 'Controller operating mode not allowed.';

	17667:
		F_ADSErrorCodeExt := 'The value for the percentage weighting of the velocity pre-control is not allowed. The parameter is pre-set to 1.0 (100%) as standard.';

	17668:
		F_ADSErrorCodeExt := 'The value for the activation of the following error monitoring is not allowed.';

	17669:
		F_ADSErrorCodeExt := 'The value for the activation of the following error monitoring (velocity) is not allowed.';

	17670:
		F_ADSErrorCodeExt := 'The value for the following error window (maximum allowable following error) is not allowed.';

	17671:
		F_ADSErrorCodeExt := 'The value for the following error filter time (position) is not allowed.';

	17672:
		F_ADSErrorCodeExt := 'The value for the following error window (velocity) is not allowed.';

	17673:
		F_ADSErrorCodeExt := 'The value for the following error filter time (velocity) is not allowed.';

	17674:
		F_ADSErrorCodeExt := '“Controller Output Limitation” Improper';

	17680:
		F_ADSErrorCodeExt := 'Proportional gain Kv or Kp (controller) not allowed.';

	17681:
		F_ADSErrorCodeExt := 'Integral-action time Tn (controller) not allowed.';

	17682:
		F_ADSErrorCodeExt := 'Derivative action time Tv (controller) not allowed.';

	17683:
		F_ADSErrorCodeExt := 'Damping time Td (controller) not allowed.';

	17684:
		F_ADSErrorCodeExt := 'Activation of the automatic offset compensation not allowed.';

	17685:
		F_ADSErrorCodeExt := 'Additional proportional gain Kv or Kp (controller) not allowed.';

	17686:
		F_ADSErrorCodeExt := 'Reference velocity for additional proportional gain Kv or Kp (controller) not allowed.';

	17687:
		F_ADSErrorCodeExt := 'Proportional gain Pa (proportion) not allowed.';

	17688:
		F_ADSErrorCodeExt := 'Proportional gain Kv (velocity controller) not allowed.';

	17689:
		F_ADSErrorCodeExt := 'Reset time Tn (velocity controller) not allowed.';

	17690:
		F_ADSErrorCodeExt := 'Reserved';

	17691:
		F_ADSErrorCodeExt := 'Reserved';

	17692:
		F_ADSErrorCodeExt := 'Velocity Filter Time” Improper';

	17693:
		F_ADSErrorCodeExt := 'Dead zone not allowed.';

	17695:
		F_ADSErrorCodeExt := 'Proportionality Factor Kcp” Improper.';

	17696:
		F_ADSErrorCodeExt := 'Rate time Tv (velocity controller) not allowed.';

	17697:
		F_ADSErrorCodeExt := 'Damping time Td (velocity controller) not allowed.';

	17698:
		F_ADSErrorCodeExt := 'Limitation of the I Part” Improper.';

	17699:
		F_ADSErrorCodeExt := 'Limitation of the D Part” Improper.';

	17700:
		F_ADSErrorCodeExt := 'Parameter “Switching Off the I Part During Motion” is Improper.';

	17701:
		F_ADSErrorCodeExt := 'Parameter “Filter Time for P-T2 Filter” Improper.';

	17702:
		F_ADSErrorCodeExt := 'Velocity Observer: “Parameterized Mode” is Improper.';

	17703:
		F_ADSErrorCodeExt := 'Velocity Observer: “Motor Torque Constant Kt or Kf” is Improper.';

	17704:
		F_ADSErrorCodeExt := 'Velocity Observer: “Motor Moment of Inertia JM” is Improper.';

	17705:
		F_ADSErrorCodeExt := 'Velocity Observer: “Band Width f0” is Improper.';

	17706:
		F_ADSErrorCodeExt := 'Velocity Observer: “Correction Factor kc” is Improper.';

	17707:
		F_ADSErrorCodeExt := 'Velocity Observer: “Time Constant T for First Order Filter” is Improper.';

	17708:
		F_ADSErrorCodeExt := 'Velocity Observer: “Amplitude Damping d for Second Order Filter” is Improper.';

	17709:
		F_ADSErrorCodeExt := 'Velocity Observer: “Frequency fHP or Frequency fTP for Filters of Second Order” is Improper.';

	17728:
		F_ADSErrorCodeExt := 'Controller has not been initialized.';

	17729:
		F_ADSErrorCodeExt := 'Controller does not know its axis, or the axis address has not been initialized.';

	17730:
		F_ADSErrorCodeExt := 'Controller does not know its drive, or the drive address has not been initialized.';

	17744:
		F_ADSErrorCodeExt := 'Following error monitoring (position). A following error exceedance has occurred';

	17745:
		F_ADSErrorCodeExt := 'Following error monitoring (velocity). A velocity following error exceedance has occurred';

	17824:
		F_ADSErrorCodeExt := 'CONTROLERR_RANGE_AREA_ASIDE';

	17825:
		F_ADSErrorCodeExt := 'CONTROLERR_RANGE_AREA_BSIDE';

	17826:
		F_ADSErrorCodeExt := 'CONTROLERR_RANGE_QNENN';

	17827:
		F_ADSErrorCodeExt := 'CONTROLERR_RANGE_PNENN';

	17828:
		F_ADSErrorCodeExt := 'CONTROLERR_RANGE_AXISIDPRESP0';

		// NC - Drive Error Codes 

	// 17920 - 18005
	17920:
		F_ADSErrorCodeExt := 'Drive ID not allowed.';

	17921:
		F_ADSErrorCodeExt := 'Drive type not allowed.';

	17922:
		F_ADSErrorCodeExt := 'Drive operation mode not allowed.';

	17923:
		F_ADSErrorCodeExt := 'Motor polarity inverted?.';

	17924:
		F_ADSErrorCodeExt := 'The value for the drift compensation (DAC offset) is not allowed.';

	17925:
		F_ADSErrorCodeExt := 'The value for the reference velocity (also called velocity pre-control) is not allowed.';

	17926:
		F_ADSErrorCodeExt := 'The value for the reference output in percent is not allowed. The value 1.0 (100 %) usually corresponds to a voltage of 10.0 V.';

	17927:
		F_ADSErrorCodeExt := 'The value for the quadrant compensation factor is not allowed.';

	17928:
		F_ADSErrorCodeExt := 'The value for the velocity reference point in percent is not allowed. The value 1.0 corresponds to 100 percent.';

	17929:
		F_ADSErrorCodeExt := 'The value for the output reference point in percent is not allowed. The value 1.0 corresponds to 100 percent.';

	17930:
		F_ADSErrorCodeExt := 'The value for the minimum and/or maximum drive output limit is not allowed.';

	17931:
		F_ADSErrorCodeExt := 'Parameter "Maximum value for output" is not allowed';

	17932:
		F_ADSErrorCodeExt := 'Parameter "Internal Drive Control Word" is not allowed';

	17933:
		F_ADSErrorCodeExt := 'Parameter "Internal timer for RESET behavior Drive" is not allowed';

	17934:
		F_ADSErrorCodeExt := 'Parameter "Master Motion Controller ID" is not allowed';

	17935:
		F_ADSErrorCodeExt := 'Drive torque output scaling not allowed.';

	17936:
		F_ADSErrorCodeExt := 'Drive velocity output scaling not allowed.';

	17937:
		F_ADSErrorCodeExt := 'Profi Drive DSC proportional gain Kpc (controller) not allowed.';

	17938:
		F_ADSErrorCodeExt := 'The value for the table ID is not allowed.';

	17939:
		F_ADSErrorCodeExt := 'The value is not allowed as the table interpolation type.';

	17940:
		F_ADSErrorCodeExt := 'The value is not allowed as an output offset in percent (+/- 1.0).';

	17941:
		F_ADSErrorCodeExt := 'Profi Drive DSC scaling for calculation of "Xerr" (controller) not allowed.';

	17942:
		F_ADSErrorCodeExt := 'The value is not allowed as drive acceleration/deceleration output scaling.';

	17943:
		F_ADSErrorCodeExt := 'The value is not allowed as drive position output scaling.';

	17944:
		F_ADSErrorCodeExt := 'Parameter "Dead time compensation mode" (Motion Controller) is invalid';

	17945:
		F_ADSErrorCodeExt := 'Parameter "Control bits of the dead time compensation" (Motion Controller) is invalid';

	17946:
		F_ADSErrorCodeExt := 'Parameter "time shift of dead time compensation mode" (Motion Controller) is invalid';

	17947:
		F_ADSErrorCodeExt := 'Parameter "Output delay velocity interface Motion Controller" is invalid';

	17948:
		F_ADSErrorCodeExt := 'Drive filter type not allowed for command variable filter for the output position.';

	17949:
		F_ADSErrorCodeExt := 'Drive filter time not allowed for command variable filter for the output position.';

	17950:
		F_ADSErrorCodeExt := 'The value is not allowed as a drive filter order (P-Tn) for the smoothing of the output position (command variable filter for the set position).';

	17952:
		F_ADSErrorCodeExt := 'Bit mask for stepper motor cycle not allowed.';

	17953:
		F_ADSErrorCodeExt := 'Bit mask for stepper motor holding current not allowed.';

	17954:
		F_ADSErrorCodeExt := 'Scaling factor for actual torque (actual current) not allowed.';

	17955:
		F_ADSErrorCodeExt := 'Filter time for actual torque is not allowed.';

	17956:
		F_ADSErrorCodeExt := 'Filter time for the temporal derivation of the actual torque is not allowed.';

	17957:
		F_ADSErrorCodeExt := 'Parameter "Drive operation mode" is invalid';

	17958:
		F_ADSErrorCodeExt := 'Motion Controller function is not supported';

	17959:
		F_ADSErrorCodeExt := 'The activation of the drive operation mode failed, because another object with OID… is already using this interface.';

	17960:
		F_ADSErrorCodeExt := 'Drive operation mode changeover is not configured or the desired drive operation mode cannot be found';

	17961:
		F_ADSErrorCodeExt := 'Feedback drive operation mode changeover';

	17968:
		F_ADSErrorCodeExt := 'Overtemperature" Overtemperature was detected or reported in the drive or terminal.';

	17969:
		F_ADSErrorCodeExt := 'Undervoltage was detected or reported in the drive or terminal.';

	17970:
		F_ADSErrorCodeExt := 'Open circuit in phase A.';

	17971:
		F_ADSErrorCodeExt := 'Open circuit in phase B.';

	17972:
		F_ADSErrorCodeExt := 'Overcurrent in phase A.';

	17973:
		F_ADSErrorCodeExt := 'Overcurrent in phase B.';

	17974:
		F_ADSErrorCodeExt := 'A torque overload (stall) was detected or reported in the drive or terminal.';

	17984:
		F_ADSErrorCodeExt := 'Drive has not been initialized.';

	17985:
		F_ADSErrorCodeExt := 'Drive does not know its axis, or the axis address has not been initialized.';

	17986:
		F_ADSErrorCodeExt := 'Drive has no valid I/O input address in the process image.';

	17987:
		F_ADSErrorCodeExt := 'Drive has no valid I/O output address in the process image.';

	18000:
		F_ADSErrorCodeExt := 'The drive hardware is not ready for operation.';

	18001:
		F_ADSErrorCodeExt := 'Error in the cyclic communication of the drive (Life Counter). Reasons for this could be an interrupted fieldbus or a drive that is in the error state.';

	18002:
		F_ADSErrorCodeExt := 'Changing the table ID when active controller enable is not allowed.';

	18005:
		F_ADSErrorCodeExt := 'Invalid I/O data for more than "n" continuous NC cycles.';

		// NC - Table Error Codes

	// 18944 - 18981
	18944:
		F_ADSErrorCodeExt := 'Table ID not allowed.';

	18945:
		F_ADSErrorCodeExt := 'Table type not allowed.';

	18946:
		F_ADSErrorCodeExt := 'Number of lines in the table not allowed.';

	18947:
		F_ADSErrorCodeExt := 'Number of columns in the table is not allowed.';

	18948:
		F_ADSErrorCodeExt := 'Step size (position delta) not allowed.';

	18949:
		F_ADSErrorCodeExt := 'Period not allowed.';

	18950:
		F_ADSErrorCodeExt := 'Table is not monotonic.';

	18951:
		F_ADSErrorCodeExt := 'Table sub type is not allowed.';

	18952:
		F_ADSErrorCodeExt := 'Table interpolation type is not allowed.';

	18953:
		F_ADSErrorCodeExt := 'The table main type is unknown or otherwise the table class (slave type) do not match up to the table main type.';

	18960:
		F_ADSErrorCodeExt := 'Table has not been initialized.';

	18961:
		F_ADSErrorCodeExt := 'Table could not be created, since there is not enough memory.';

	18962:
		F_ADSErrorCodeExt := 'The function has not been implemented, or cannot be executed, for the present type of table.';

	18963:
		F_ADSErrorCodeExt := 'The start line index or the stop line index to be used for read or write access to the table is not allowed.';

	18964:
		F_ADSErrorCodeExt := 'The start column index or the stop column index to be used for read or write access to the table in not allowed.';

	18965:
		F_ADSErrorCodeExt := 'The number of lines to be read from or written to the table is not allowed.';

	18966:
		F_ADSErrorCodeExt := 'The number of columns to be read from or written to the table is not allowed.';

	18967:
		F_ADSErrorCodeExt := 'The entries in the table header are inconsistent, e.g. the validity range is empty.';

	18968:
		F_ADSErrorCodeExt := 'The slave master position is outside the table values for the master.';

	18969:
		F_ADSErrorCodeExt := 'Solo table underflow. The slave master position is outside the table values for the master.';

	18970:
		F_ADSErrorCodeExt := 'Solo table overflow. The slave master position is outside the table values for the master.';

	18971:
		F_ADSErrorCodeExt := 'Incorrect execution mode.';

	18972:
		F_ADSErrorCodeExt := 'Impermissible parameter. The Fifo parameter is not allowed.';

	18973:
		F_ADSErrorCodeExt := 'Fifo is empty.';

	18974:
		F_ADSErrorCodeExt := 'Fifo is full.';

	18975:
		F_ADSErrorCodeExt := 'Point-Index of Motion Function invalid.';

	18976:
		F_ADSErrorCodeExt := 'No diagonalisation of  matrix. The spline can not be calculated.';

	18977:
		F_ADSErrorCodeExt := 'The number of points of a cubic spline has to be greater than two.';

	18978:
		F_ADSErrorCodeExt := 'Fifo must not be overwritten.';

	18979:
		F_ADSErrorCodeExt := 'Insufficient number of Motion Function points.';

	18981:
		F_ADSErrorCodeExt := 'A periodic position table must start with a master position zero.';

		// NC - NC-PLC Error Codes

	// 19200 - 19395
	19200:
		F_ADSErrorCodeExt := 'The axis was stopped during travel to the target position.';

	19201:
		F_ADSErrorCodeExt := 'Axis cannot be started. Error, or busy, or protected, or not ready for operation.';

	19202:
		F_ADSErrorCodeExt := 'No target position control, and no position range control permitted.';

	19203:
		F_ADSErrorCodeExt := 'The position and velocity can only be restarted while the axis is physically in motion.';

	19204:
		F_ADSErrorCodeExt := 'Invalid mode. Invalide Direction with MC_MoveModulo, or inactive axis parameter "Position Correction" with MC_BacklashCompensation.';

	19205:
		F_ADSErrorCodeExt := 'Command not permitted. Direction not specified, or read/write parameter type mismatch.';

	19206:
		F_ADSErrorCodeExt := 'Parameter incorrect. Override outside bounds, or read/write parameter type mismatch.';

